LIN {X 0,Y 636.346,Z 292.016,A -85,B 0,C 180,E1 -5612.399,E2 -5612.399} C_VEL
LIN {X 0,Y 638.577,Z 243.118,A -85,B 0,C 180,E1 -5615.474,E2 -5615.474} C_VEL
LIN {X 0,Y 628.677,Z 217.087,A -85,B 0,C 180,E1 -5617.846,E2 -5617.846} C_VEL
LIN {X 0,Y 624.895,Z 207.391,A -85,B 0,C 180,E1 -5618.774,E2 -5618.774} C_VEL
LIN {X 0,Y 624.9,Z 207.391,A -85,B 0,C 180,E1 -5622.101,E2 -5622.101} C_VEL
LIN {X 0,Y 624.949,Z 207.381,A -85,B 0,C 180,E1 -5625.136,E2 -5625.136} C_VEL
LIN {X 0,Y 624.933,Z 207.387,A -85,B 0,C 180,E1 -5628.349,E2 -5628.349} C_VEL
LIN {X 0,Y 624.928,Z 207.584,A -85,B 0,C 180,E1 -5630.263,E2 -5630.263} C_VEL
LIN {X 0,Y 626.015,Z 210.6,A -85,B 0,C 180,E1 -5630.528,E2 -5630.528} C_VEL
LIN {X 0,Y 632.721,Z 226.25,A -85,B 0,C 180,E1 -5632.053,E2 -5632.053} C_VEL
LIN {X 0,Y 640.273,Z 245.58,A -85,B 0,C 180,E1 -5633.993,E2 -5633.993} C_VEL
LIN {X 0,Y 640.705,Z 247.691,A -85,B 0,C 180,E1 -5634.181,E2 -5634.181} C_VEL
LIN {X 0,Y 639.221,Z 289.191,A -85,B 0,C 180,E1 -5637.233,E2 -5637.233} C_VEL
LIN {X 0,Y 638.897,Z 318.308,A -85,B 0,C 180,E1 -5639.227,E2 -5639.227} C_VEL
LIN {X 0,Y 639.099,Z 324.989,A -85,B 0,C 180,E1 -5639.637,E2 -5639.637} C_VEL
LIN {X 0,Y 639.536,Z 329.306,A -85,B 0,C 180,E1 -5639.718,E2 -5639.718} C_VEL
LIN {X 0,Y 637.723,Z 440.539,A -85,B 0,C 180,E1 -5641.138,E2 -5641.138} C_VEL
LIN {X 0,Y 634.236,Z 617.38,A -85,B 0,C 180,E1 -5643.602,E2 -5643.602} C_VEL
LIN {X 0,Y 633.701,Z 640.001,A -85,B 0,C 180,E1 -5644.083,E2 -5644.083} C_VEL
LIN {X 0,Y 632.964,Z 662.226,A -85,B 0,C 180,E1 -5644.728,E2 -5644.728} C_VEL
LIN {X 0,Y 632.12,Z 684.246,A -85,B 0,C 180,E1 -5645.551,E2 -5645.551} C_VEL
LIN {X 0,Y 631.255,Z 703.32,A -85,B 0,C 180,E1 -5646.425,E2 -5646.425} C_VEL
LIN {X 0,Y 630.24,Z 722.986,A -85,B 0,C 180,E1 -5647.52,E2 -5647.52} C_VEL
LIN {X 0,Y 629.208,Z 740.926,A -85,B 0,C 180,E1 -5648.708,E2 -5648.708} C_VEL
LIN {X 0,Y 628.174,Z 758.568,A -85,B 0,C 180,E1 -5650.085,E2 -5650.085} C_VEL
LIN {X 0,Y 627.247,Z 774.118,A -85,B 0,C 180,E1 -5651.505,E2 -5651.505} C_VEL
LIN {X 0,Y 626.389,Z 788.139,A -85,B 0,C 180,E1 -5653.015,E2 -5653.015} C_VEL
LIN {X 0,Y 625.582,Z 802.216,A -85,B 0,C 180,E1 -5654.804,E2 -5654.804} C_VEL
LIN {X 0,Y 624.988,Z 813.341,A -85,B 0,C 180,E1 -5656.492,E2 -5656.492} C_VEL
LIN {X 0,Y 624.565,Z 822.244,A -85,B 0,C 180,E1 -5658.081,E2 -5658.081} C_VEL
LIN {X 0,Y 624.211,Z 832.3,A -85,B 0,C 180,E1 -5660.224,E2 -5660.224} C_VEL
LIN {X 0,Y 624.048,Z 838.961,A -85,B 0,C 180,E1 -5661.987,E2 -5661.987} C_VEL
LIN {X 0,Y 623.969,Z 843.988,A -85,B 0,C 180,E1 -5663.652,E2 -5663.652} C_VEL
LIN {X 0,Y 623.918,Z 847.629,A -85,B 0,C 180,E1 -5665.22,E2 -5665.22} C_VEL
LIN {X 0,Y 623.903,Z 850.253,A -85,B 0,C 180,E1 -5666.807,E2 -5666.807} C_VEL
LIN {X 0,Y 623.908,Z 851.807,A -85,B 0,C 180,E1 -5668.347,E2 -5668.347} C_VEL
LIN {X 0,Y 623.919,Z 852.393,A -85,B 0,C 180,E1 -5670,E2 -5670} C_VEL
LIN {X 0,Y 623.906,Z 851.865,A -85,B 0,C 180,E1 -5671.653,E2 -5671.653} C_VEL
LIN {X 0,Y 623.901,Z 850.34,A -85,B 0,C 180,E1 -5673.215,E2 -5673.215} C_VEL
LIN {X 0,Y 623.92,Z 847.804,A -85,B 0,C 180,E1 -5674.78,E2 -5674.78} C_VEL
LIN {X 0,Y 623.969,Z 844.223,A -85,B 0,C 180,E1 -5676.348,E2 -5676.348} C_VEL
LIN {X 0,Y 624.029,Z 839.56,A -85,B 0,C 180,E1 -5677.92,E2 -5677.92} C_VEL
LIN {X 0,Y 624.164,Z 833.767,A -85,B 0,C 180,E1 -5679.497,E2 -5679.497} C_VEL
LIN {X 0,Y 624.432,Z 825.538,A -85,B 0,C 180,E1 -5681.359,E2 -5681.359} C_VEL
LIN {X 0,Y 624.9,Z 815.025,A -85,B 0,C 180,E1 -5683.321,E2 -5683.321} C_VEL
LIN {X 0,Y 625.468,Z 804.166,A -85,B 0,C 180,E1 -5685.009,E2 -5685.009} C_VEL
LIN {X 0,Y 626.179,Z 791.739,A -85,B 0,C 180,E1 -5686.646,E2 -5686.646} C_VEL
LIN {X 0,Y 627.018,Z 777.74,A -85,B 0,C 180,E1 -5688.213,E2 -5688.213} C_VEL
LIN {X 0,Y 627.946,Z 762.367,A -85,B 0,C 180,E1 -5689.68,E2 -5689.68} C_VEL
LIN {X 0,Y 628.974,Z 745.456,A -85,B 0,C 180,E1 -5691.056,E2 -5691.056} C_VEL
LIN {X 0,Y 629.98,Z 727.417,A -85,B 0,C 180,E1 -5692.292,E2 -5692.292} C_VEL
LIN {X 0,Y 630.985,Z 708.54,A -85,B 0,C 180,E1 -5693.388,E2 -5693.388} C_VEL
LIN {X 0,Y 631.859,Z 689.995,A -85,B 0,C 180,E1 -5694.295,E2 -5694.295} C_VEL
LIN {X 0,Y 632.742,Z 669.051,A -85,B 0,C 180,E1 -5695.13,E2 -5695.13} C_VEL
LIN {X 0,Y 633.413,Z 648.623,A -85,B 0,C 180,E1 -5695.774,E2 -5695.774} C_VEL
LIN {X 0,Y 634.025,Z 626.542,A -85,B 0,C 180,E1 -5696.308,E2 -5696.308} C_VEL
LIN {X 0,Y 634.453,Z 605.1,A -85,B 0,C 180,E1 -5696.679,E2 -5696.679} C_VEL
LIN {X 0,Y 638.365,Z 407.202,A -85,B 0,C 180,E1 -5699.392,E2 -5699.392} C_VEL
LIN {X 0,Y 639.37,Z 326.363,A -85,B 0,C 180,E1 -5700.421,E2 -5700.421} C_VEL
LIN {X 0,Y 639.015,Z 324.152,A -85,B 0,C 180,E1 -5700.489,E2 -5700.489} C_VEL
LIN {X 0,Y 639.079,Z 296.354,A -85,B 0,C 180,E1 -5702.35,E2 -5702.35} C_VEL
LIN {X 0,Y 640.388,Z 256.622,A -85,B 0,C 180,E1 -5705.253,E2 -5705.253} C_VEL
LIN {X 0,Y 640.643,Z 246.721,A -85,B 0,C 180,E1 -5705.976,E2 -5705.976} C_VEL
LIN {X 0,Y 633.821,Z 228.869,A -85,B 0,C 180,E1 -5707.781,E2 -5707.781} C_VEL
LIN {X 0,Y 627.274,Z 213.434,A -85,B 0,C 180,E1 -5709.294,E2 -5709.294} C_VEL
LIN {X 0,Y 624.952,Z 207.388,A -85,B 0,C 180,E1 -5709.871,E2 -5709.871} C_VEL
LIN {X 0,Y 624.924,Z 207.385,A -85,B 0,C 180,E1 -5713.012,E2 -5713.012} C_VEL
LIN {X 0,Y 624.946,Z 207.377,A -85,B 0,C 180,E1 -5716.149,E2 -5716.149} C_VEL
LIN {X 0,Y 624.928,Z 207.382,A -85,B 0,C 180,E1 -5719.246,E2 -5719.246} C_VEL
LIN {X 0,Y 624.947,Z 207.376,A -85,B 0,C 180,E1 -5722.371,E2 -5722.371} C_VEL
LIN {X 0,Y 624.94,Z 207.389,A -85,B 0,C 180,E1 -5725.501,E2 -5725.501} C_VEL
LIN {X 0,Y 624.947,Z 207.379,A -85,B 0,C 180,E1 -5728.776,E2 -5728.776} C_VEL
LIN {X 0,Y 624.945,Z 207.373,A -85,B 0,C 180,E1 -5731.94,E2 -5731.94} C_VEL
LIN {X 0,Y 624.937,Z 207.381,A -85,B 0,C 180,E1 -5735.12,E2 -5735.12} C_VEL
LIN {X 0,Y 624.937,Z 207.383,A -85,B 0,C 180,E1 -5738.21,E2 -5738.21} C_VEL
LIN {X 0,Y 624.937,Z 207.371,A -85,B 0,C 180,E1 -5741.337,E2 -5741.337} C_VEL
LIN {X 0,Y 624.934,Z 207.381,A -85,B 0,C 180,E1 -5744.407,E2 -5744.407} C_VEL
LIN {X 0,Y 624.941,Z 207.366,A -85,B 0,C 180,E1 -5747.526,E2 -5747.526} C_VEL
LIN {X 0,Y 624.942,Z 207.38,A -85,B 0,C 180,E1 -5750.7,E2 -5750.7} C_VEL
LIN {X 0,Y 624.943,Z 207.365,A -85,B 0,C 180,E1 -5753.938,E2 -5753.938} C_VEL
LIN {X 0,Y 624.947,Z 207.38,A -85,B 0,C 180,E1 -5757.157,E2 -5757.157} C_VEL
LIN {X 0,Y 624.923,Z 207.363,A -85,B 0,C 180,E1 -5760.275,E2 -5760.275} C_VEL
LIN {X 0,Y 624.946,Z 207.381,A -85,B 0,C 180,E1 -5763.394,E2 -5763.394} C_VEL
LIN {X 0,Y 624.919,Z 207.364,A -85,B 0,C 180,E1 -5766.523,E2 -5766.523} C_VEL
LIN {X 0,Y 624.949,Z 207.381,A -85,B 0,C 180,E1 -5769.671,E2 -5769.671} C_VEL
LIN {X 0,Y 624.924,Z 207.382,A -85,B 0,C 180,E1 -5772.756,E2 -5772.756} C_VEL
LIN {X 0,Y 624.942,Z 207.385,A -85,B 0,C 180,E1 -5775.974,E2 -5775.974} C_VEL
LIN {X 0,Y 624.946,Z 207.377,A -85,B 0,C 180,E1 -5779.147,E2 -5779.147} C_VEL
LIN {X 0,Y 624.916,Z 207.388,A -85,B 0,C 180,E1 -5782.358,E2 -5782.358} C_VEL
LIN {X 0,Y 624.953,Z 207.381,A -85,B 0,C 180,E1 -5785.391,E2 -5785.391} C_VEL
LIN {X 0,Y 624.91,Z 207.385,A -85,B 0,C 180,E1 -5788.546,E2 -5788.546} C_VEL
LIN {X 0,Y 624.957,Z 207.381,A -85,B 0,C 180,E1 -5791.546,E2 -5791.546} C_VEL
LIN {X 0,Y 624.906,Z 207.388,A -85,B 0,C 180,E1 -5794.671,E2 -5794.671} C_VEL
LIN {X 0,Y 624.957,Z 207.38,A -85,B 0,C 180,E1 -5797.791,E2 -5797.791} C_VEL
LIN {X 0,Y 624.903,Z 207.389,A -85,B 0,C 180,E1 -5800.814,E2 -5800.814} C_VEL
LIN {X 0,Y 624.95,Z 207.462,A -85,B 0,C 180,E1 -5803.387,E2 -5803.387} C_VEL
LIN {X 0,Y 626.289,Z 210.904,A -85,B 0,C 180,E1 -5803.733,E2 -5803.733} C_VEL
LIN {X 0,Y 627.344,Z 212.887,A -85,B 0,C 180,E1 -5803.957,E2 -5803.957} C_VEL
LIN {X 0,Y 638.156,Z 234.423,A -85,B 0,C 180,E1 -5806.246,E2 -5806.246} C_VEL
LIN {X 0,Y 647.363,Z 253.935,A -85,B 0,C 180,E1 -5808.145,E2 -5808.145} C_VEL
LIN {X 0,Y 644.416,Z 304.648,A -85,B 0,C 180,E1 -5810.782,E2 -5810.782} C_VEL
LIN {X 0,Y 646.898,Z 323.157,A -85,B 0,C 180,E1 -5811.205,E2 -5811.205} C_VEL
LIN {X 0,Y 644.169,Z 514.087,A -85,B 0,C 180,E1 -5813.627,E2 -5813.627} C_VEL
LIN {X 0,Y 641.865,Z 692.934,A -85,B 0,C 180,E1 -5815.853,E2 -5815.853} C_VEL
LIN {X 0,Y 641.079,Z 718.1,A -85,B 0,C 180,E1 -5816.326,E2 -5816.326} C_VEL
LIN {X 0,Y 640.186,Z 739.868,A -85,B 0,C 180,E1 -5816.869,E2 -5816.869} C_VEL
LIN {X 0,Y 638.916,Z 765.321,A -85,B 0,C 180,E1 -5817.682,E2 -5817.682} C_VEL
LIN {X 0,Y 637.689,Z 787.238,A -85,B 0,C 180,E1 -5818.539,E2 -5818.539} C_VEL
LIN {X 0,Y 636.241,Z 810.546,A -85,B 0,C 180,E1 -5819.631,E2 -5819.631} C_VEL
LIN {X 0,Y 634.874,Z 830.591,A -85,B 0,C 180,E1 -5820.724,E2 -5820.724} C_VEL
LIN {X 0,Y 633.292,Z 852.909,A -85,B 0,C 180,E1 -5822.138,E2 -5822.138} C_VEL
LIN {X 0,Y 632.055,Z 867.818,A -85,B 0,C 180,E1 -5823.252,E2 -5823.252} C_VEL
LIN {X 0,Y 630.517,Z 886.159,A -85,B 0,C 180,E1 -5824.798,E2 -5824.798} C_VEL
LIN {X 0,Y 629.035,Z 903.822,A -85,B 0,C 180,E1 -5826.518,E2 -5826.518} C_VEL
LIN {X 0,Y 627.829,Z 919.315,A -85,B 0,C 180,E1 -5828.218,E2 -5828.218} C_VEL
LIN {X 0,Y 626.714,Z 934.515,A -85,B 0,C 180,E1 -5830.133,E2 -5830.133} C_VEL
LIN {X 0,Y 625.867,Z 947.149,A -85,B 0,C 180,E1 -5831.945,E2 -5831.945} C_VEL
LIN {X 0,Y 625.118,Z 960.283,A -85,B 0,C 180,E1 -5834.126,E2 -5834.126} C_VEL
LIN {X 0,Y 624.657,Z 970.018,A -85,B 0,C 180,E1 -5836.013,E2 -5836.013} C_VEL
LIN {X 0,Y 624.293,Z 979.836,A -85,B 0,C 180,E1 -5838.264,E2 -5838.264} C_VEL
LIN {X 0,Y 624.094,Z 986.816,A -85,B 0,C 180,E1 -5840.222,E2 -5840.222} C_VEL
LIN {X 0,Y 623.952,Z 993.243,A -85,B 0,C 180,E1 -5842.449,E2 -5842.449} C_VEL
LIN {X 0,Y 623.905,Z 997.655,A -85,B 0,C 180,E1 -5844.574,E2 -5844.574} C_VEL
LIN {X 0,Y 623.91,Z 1000.464,A -85,B 0,C 180,E1 -5846.509,E2 -5846.509} C_VEL
LIN {X 0,Y 623.909,Z 1002.214,A -85,B 0,C 180,E1 -5848.806,E2 -5848.806} C_VEL
LIN {X 0,Y 623.885,Z 1002.327,A -85,B 0,C 180,E1 -5850.735,E2 -5850.735} C_VEL
LIN {X 0,Y 623.889,Z 1001.292,A -85,B 0,C 180,E1 -5852.664,E2 -5852.664} C_VEL
LIN {X 0,Y 623.901,Z 998.451,A -85,B 0,C 180,E1 -5854.965,E2 -5854.965} C_VEL
LIN {X 0,Y 623.959,Z 994.689,A -85,B 0,C 180,E1 -5856.903,E2 -5856.903} C_VEL
LIN {X 0,Y 624.042,Z 988.934,A -85,B 0,C 180,E1 -5859.127,E2 -5859.127} C_VEL
LIN {X 0,Y 624.217,Z 981.602,A -85,B 0,C 180,E1 -5861.27,E2 -5861.27} C_VEL
LIN {X 0,Y 624.519,Z 973.532,A -85,B 0,C 180,E1 -5863.235,E2 -5863.235} C_VEL
LIN {X 0,Y 624.996,Z 962.86,A -85,B 0,C 180,E1 -5865.401,E2 -5865.401} C_VEL
LIN {X 0,Y 625.602,Z 951.969,A -85,B 0,C 180,E1 -5867.294,E2 -5867.294} C_VEL
LIN {X 0,Y 626.517,Z 937.317,A -85,B 0,C 180,E1 -5869.485,E2 -5869.485} C_VEL
LIN {X 0,Y 627.462,Z 924.012,A -85,B 0,C 180,E1 -5871.215,E2 -5871.215} C_VEL
LIN {X 0,Y 628.838,Z 906.301,A -85,B 0,C 180,E1 -5873.225,E2 -5873.225} C_VEL
LIN {X 0,Y 630.114,Z 890.795,A -85,B 0,C 180,E1 -5874.767,E2 -5874.767} C_VEL
LIN {X 0,Y 631.805,Z 870.854,A -85,B 0,C 180,E1 -5876.506,E2 -5876.506} C_VEL
LIN {X 0,Y 633.107,Z 855.309,A -85,B 0,C 180,E1 -5877.693,E2 -5877.693} C_VEL
LIN {X 0,Y 634.055,Z 841.543,A -85,B 0,C 180,E1 -5878.595,E2 -5878.595} C_VEL
LIN {X 0,Y 635.449,Z 820.222,A -85,B 0,C 180,E1 -5879.817,E2 -5879.817} C_VEL
LIN {X 0,Y 636.697,Z 797.901,A -85,B 0,C 180,E1 -5880.899,E2 -5880.899} C_VEL
LIN {X 0,Y 637.906,Z 775.285,A -85,B 0,C 180,E1 -5881.835,E2 -5881.835} C_VEL
LIN {X 0,Y 638.944,Z 751.93,A -85,B 0,C 180,E1 -5882.623,E2 -5882.623} C_VEL
LIN {X 0,Y 639.847,Z 727.921,A -85,B 0,C 180,E1 -5883.28,E2 -5883.28} C_VEL
LIN {X 0,Y 640.534,Z 703.096,A -85,B 0,C 180,E1 -5883.781,E2 -5883.781} C_VEL
LIN {X 0,Y 640.998,Z 677.434,A -85,B 0,C 180,E1 -5884.144,E2 -5884.144} C_VEL
LIN {X 0,Y 642.199,Z 471.258,A -85,B 0,C 180,E1 -5886.503,E2 -5886.503} C_VEL
LIN {X 0,Y 643.617,Z 320.826,A -85,B 0,C 180,E1 -5888.348,E2 -5888.348} C_VEL
LIN {X 0,Y 642.214,Z 312.028,A -85,B 0,C 180,E1 -5888.548,E2 -5888.548} C_VEL
LIN {X 0,Y 644.812,Z 281.295,A -85,B 0,C 180,E1 -5890.288,E2 -5890.288} C_VEL
LIN {X 0,Y 648.358,Z 254.707,A -85,B 0,C 180,E1 -5891.95,E2 -5891.95} C_VEL
LIN {X 0,Y 645.178,Z 246.171,A -85,B 0,C 180,E1 -5893.117,E2 -5893.117} C_VEL
LIN {X 0,Y 642.634,Z 240.116,A -85,B 0,C 180,E1 -5894.191,E2 -5894.191} C_VEL
LIN {X 0,Y 641.16,Z 236.75,A -85,B 0,C 180,E1 -5894.947,E2 -5894.947} C_VEL
LIN {X 0,Y 639.826,Z 233.597,A -85,B 0,C 180,E1 -5895.832,E2 -5895.832} C_VEL
LIN {X 0,Y 638.452,Z 230.647,A -85,B 0,C 180,E1 -5897.302,E2 -5897.302} C_VEL
LIN {X 0,Y 638.405,Z 229.859,A -85,B 0,C 180,E1 -5898.268,E2 -5898.268} C_VEL
LIN {X 0,Y 638.414,Z 231.106,A -85,B 0,C 180,E1 -5899.342,E2 -5899.342} C_VEL
LIN {X 0,Y 639.781,Z 233.899,A -85,B 0,C 180,E1 -5900.68,E2 -5900.68} C_VEL
LIN {X 0,Y 641.35,Z 238.172,A -85,B 0,C 180,E1 -5901.791,E2 -5901.791} C_VEL
LIN {X 0,Y 643.354,Z 243.746,A -85,B 0,C 180,E1 -5902.873,E2 -5902.873} C_VEL
LIN {X 0,Y 645.653,Z 251.249,A -85,B 0,C 180,E1 -5903.999,E2 -5903.999} C_VEL
LIN {X 0,Y 641.269,Z 281.594,A -85,B 0,C 180,E1 -5906.283,E2 -5906.283} C_VEL
LIN {X 0,Y 637.312,Z 322.129,A -85,B 0,C 180,E1 -5909.115,E2 -5909.115} C_VEL
LIN {X 0,Y 634.413,Z 366.282,A -85,B 0,C 180,E1 -5912.038,E2 -5912.038} C_VEL
LIN {X 0,Y 631.971,Z 416.413,A -85,B 0,C 180,E1 -5915.211,E2 -5915.211} C_VEL
LIN {X 0,Y 631.044,Z 441.253,A -85,B 0,C 180,E1 -5916.72,E2 -5916.72} C_VEL
LIN {X 0,Y 635.394,Z 479.453,A -85,B 0,C 180,E1 -5917.724,E2 -5917.724} C_VEL
LIN {X 0,Y 635.961,Z 488.203,A -85,B 0,C 180,E1 -5917.919,E2 -5917.919} C_VEL
LIN {X 0,Y 632.244,Z 601.48,A -85,B 0,C 180,E1 -5919.721,E2 -5919.721} C_VEL
LIN {X 0,Y 630.407,Z 684.522,A -85,B 0,C 180,E1 -5920.982,E2 -5920.982} C_VEL
LIN {X 0,Y 629.845,Z 705.803,A -85,B 0,C 180,E1 -5921.482,E2 -5921.482} C_VEL
LIN {X 0,Y 629.291,Z 724.826,A -85,B 0,C 180,E1 -5922.094,E2 -5922.094} C_VEL
LIN {X 0,Y 628.646,Z 743.951,A -85,B 0,C 180,E1 -5922.887,E2 -5922.887} C_VEL
LIN {X 0,Y 628.049,Z 760.98,A -85,B 0,C 180,E1 -5923.77,E2 -5923.77} C_VEL
LIN {X 0,Y 627.432,Z 777.32,A -85,B 0,C 180,E1 -5924.802,E2 -5924.802} C_VEL
LIN {X 0,Y 626.858,Z 791.603,A -85,B 0,C 180,E1 -5925.886,E2 -5925.886} C_VEL
LIN {X 0,Y 626.317,Z 804.831,A -85,B 0,C 180,E1 -5927.085,E2 -5927.085} C_VEL
LIN {X 0,Y 625.835,Z 816.839,A -85,B 0,C 180,E1 -5928.386,E2 -5928.386} C_VEL
LIN {X 0,Y 625.39,Z 828.124,A -85,B 0,C 180,E1 -5929.871,E2 -5929.871} C_VEL
LIN {X 0,Y 625.031,Z 837.79,A -85,B 0,C 180,E1 -5931.444,E2 -5931.444} C_VEL
LIN {X 0,Y 624.78,Z 845.408,A -85,B 0,C 180,E1 -5933.014,E2 -5933.014} C_VEL
LIN {X 0,Y 624.611,Z 851.521,A -85,B 0,C 180,E1 -5934.673,E2 -5934.673} C_VEL
LIN {X 0,Y 624.48,Z 855.819,A -85,B 0,C 180,E1 -5936.328,E2 -5936.328} C_VEL
LIN {X 0,Y 624.401,Z 858.528,A -85,B 0,C 180,E1 -5938.073,E2 -5938.073} C_VEL
LIN {X 0,Y 624.361,Z 859.436,A -85,B 0,C 180,E1 -5939.816,E2 -5939.816} C_VEL
LIN {X 0,Y 624.335,Z 858.578,A -85,B 0,C 180,E1 -5941.56,E2 -5941.56} C_VEL
LIN {X 0,Y 624.355,Z 855.951,A -85,B 0,C 180,E1 -5943.305,E2 -5943.305} C_VEL
LIN {X 0,Y 624.419,Z 851.496,A -85,B 0,C 180,E1 -5945.053,E2 -5945.053} C_VEL
LIN {X 0,Y 624.534,Z 845.462,A -85,B 0,C 180,E1 -5946.712,E2 -5946.712} C_VEL
LIN {X 0,Y 624.739,Z 837.497,A -85,B 0,C 180,E1 -5948.375,E2 -5948.375} C_VEL
LIN {X 0,Y 625.04,Z 827.956,A -85,B 0,C 180,E1 -5949.949,E2 -5949.949} C_VEL
LIN {X 0,Y 625.447,Z 816.489,A -85,B 0,C 180,E1 -5951.48,E2 -5951.48} C_VEL
LIN {X 0,Y 625.919,Z 804.267,A -85,B 0,C 180,E1 -5952.829,E2 -5952.829} C_VEL
LIN {X 0,Y 626.493,Z 790.059,A -85,B 0,C 180,E1 -5954.134,E2 -5954.134} C_VEL
LIN {X 0,Y 627.113,Z 775.015,A -85,B 0,C 180,E1 -5955.283,E2 -5955.283} C_VEL
LIN {X 0,Y 627.76,Z 758.503,A -85,B 0,C 180,E1 -5956.328,E2 -5956.328} C_VEL
LIN {X 0,Y 628.401,Z 741.33,A -85,B 0,C 180,E1 -5957.215,E2 -5957.215} C_VEL
LIN {X 0,Y 629.033,Z 723.273,A -85,B 0,C 180,E1 -5957.961,E2 -5957.961} C_VEL
LIN {X 0,Y 629.604,Z 703.456,A -85,B 0,C 180,E1 -5958.588,E2 -5958.588} C_VEL
LIN {X 0,Y 630.065,Z 683.762,A -85,B 0,C 180,E1 -5959.031,E2 -5959.031} C_VEL
LIN {X 0,Y 630.481,Z 653.884,A -85,B 0,C 180,E1 -5959.448,E2 -5959.448} C_VEL
LIN {X 0,Y 632.813,Z 483.695,A -85,B 0,C 180,E1 -5961.677,E2 -5961.677} C_VEL
LIN {X 0,Y 630.114,Z 460.538,A -85,B 0,C 180,E1 -5962.135,E2 -5962.135} C_VEL
LIN {X 0,Y 631.884,Z 406.271,A -85,B 0,C 180,E1 -5965.393,E2 -5965.393} C_VEL
LIN {X 0,Y 632.169,Z 397.972,A -85,B 0,C 180,E1 -5965.894,E2 -5965.894} C_VEL
LIN {X 0,Y 631.485,Z 391.743,A -85,B 0,C 180,E1 -5966.31,E2 -5966.31} C_VEL
LIN {X 0,Y 626.328,Z 376.015,A -85,B 0,C 180,E1 -5967.526,E2 -5967.526} C_VEL
LIN {X 0,Y 625.851,Z 370.657,A -85,B 0,C 180,E1 -5967.887,E2 -5967.887} C_VEL
LIN {X 0,Y 627.881,Z 321.996,A -85,B 0,C 180,E1 -5970.902,E2 -5970.902} C_VEL
LIN {X 0,Y 630.347,Z 269.288,A -85,B 0,C 180,E1 -5974.223,E2 -5974.223} C_VEL
LIN {X 0,Y 631.298,Z 245.645,A -85,B 0,C 180,E1 -5975.742,E2 -5975.742} C_VEL
LIN {X 0,Y 620.877,Z 218.382,A -85,B 0,C 180,E1 -5978.271,E2 -5978.271} C_VEL
LIN {X 0,Y 616.989,Z 208.38,A -85,B 0,C 180,E1 -5979.246,E2 -5979.246} C_VEL
LIN {X 0,Y 616.96,Z 208.381,A -85,B 0,C 180,E1 -5982.351,E2 -5982.351} C_VEL
LIN {X 0,Y 617.013,Z 208.37,A -85,B 0,C 180,E1 -5985.483,E2 -5985.483} C_VEL
LIN {X 0,Y 616.977,Z 208.375,A -85,B 0,C 180,E1 -5988.621,E2 -5988.621} C_VEL
LIN {X 0,Y 617.033,Z 208.453,A -85,B 0,C 180,E1 -5989.73,E2 -5989.73} C_VEL
LIN {X 0,Y 618.333,Z 211.922,A -85,B 0,C 180,E1 -5990.04,E2 -5990.04} C_VEL
LIN {X 0,Y 625.978,Z 229.789,A -85,B 0,C 180,E1 -5991.803,E2 -5991.803} C_VEL
LIN {X 0,Y 633.173,Z 248.32,A -85,B 0,C 180,E1 -5993.687,E2 -5993.687} C_VEL
LIN {X 0,Y 633.844,Z 251.207,A -85,B 0,C 180,E1 -5993.956,E2 -5993.956} C_VEL
LIN {X 0,Y 632.416,Z 295.085,A -85,B 0,C 180,E1 -5997.159,E2 -5997.159} C_VEL
LIN {X 0,Y 632.309,Z 325.01,A -85,B 0,C 180,E1 -5999.167,E2 -5999.167} C_VEL
LIN {X 0,Y 632.515,Z 327.844,A -85,B 0,C 180,E1 -5999.313,E2 -5999.313} C_VEL
LIN {X 0,Y 631.027,Z 428.42,A -85,B 0,C 180,E1 -6000.615,E2 -6000.615} C_VEL
LIN {X 0,Y 627.72,Z 572.114,A -85,B 0,C 180,E1 -6002.663,E2 -6002.663} C_VEL
LIN {X 0,Y 626.665,Z 621.823,A -85,B 0,C 180,E1 -6003.423,E2 -6003.423} C_VEL
LIN {X 0,Y 626.054,Z 644.64,A -85,B 0,C 180,E1 -6003.946,E2 -6003.946} C_VEL
LIN {X 0,Y 625.271,Z 666.522,A -85,B 0,C 180,E1 -6004.624,E2 -6004.624} C_VEL
LIN {X 0,Y 624.38,Z 687.651,A -85,B 0,C 180,E1 -6005.451,E2 -6005.451} C_VEL
LIN {X 0,Y 623.372,Z 708.562,A -85,B 0,C 180,E1 -6006.459,E2 -6006.459} C_VEL
LIN {X 0,Y 622.343,Z 727.705,A -85,B 0,C 180,E1 -6007.568,E2 -6007.568} C_VEL
LIN {X 0,Y 621.33,Z 745.237,A -85,B 0,C 180,E1 -6008.771,E2 -6008.771} C_VEL
LIN {X 0,Y 620.289,Z 761.787,A -85,B 0,C 180,E1 -6010.115,E2 -6010.115} C_VEL
LIN {X 0,Y 619.288,Z 777.907,A -85,B 0,C 180,E1 -6011.649,E2 -6011.649} C_VEL
LIN {X 0,Y 618.441,Z 791.683,A -85,B 0,C 180,E1 -6013.178,E2 -6013.178} C_VEL
LIN {X 0,Y 617.705,Z 804.058,A -85,B 0,C 180,E1 -6014.797,E2 -6014.797} C_VEL
LIN {X 0,Y 617.096,Z 815.114,A -85,B 0,C 180,E1 -6016.507,E2 -6016.507} C_VEL
LIN {X 0,Y 616.602,Z 825.387,A -85,B 0,C 180,E1 -6018.4,E2 -6018.4} C_VEL
LIN {X 0,Y 616.252,Z 834.032,A -85,B 0,C 180,E1 -6020.379,E2 -6020.379} C_VEL
LIN {X 0,Y 616.054,Z 840.215,A -85,B 0,C 180,E1 -6022.164,E2 -6022.164} C_VEL
LIN {X 0,Y 615.975,Z 844.61,A -85,B 0,C 180,E1 -6023.756,E2 -6023.756} C_VEL
LIN {X 0,Y 615.929,Z 848.876,A -85,B 0,C 180,E1 -6025.811,E2 -6025.811} C_VEL
LIN {X 0,Y 615.916,Z 851.625,A -85,B 0,C 180,E1 -6028.046,E2 -6028.046} C_VEL
LIN {X 0,Y 615.906,Z 852.387,A -85,B 0,C 180,E1 -6029.814,E2 -6029.814} C_VEL
LIN {X 0,Y 615.899,Z 851.978,A -85,B 0,C 180,E1 -6031.488,E2 -6031.488} C_VEL
LIN {X 0,Y 615.902,Z 850.572,A -85,B 0,C 180,E1 -6033.071,E2 -6033.071} C_VEL
LIN {X 0,Y 615.924,Z 848.154,A -85,B 0,C 180,E1 -6034.656,E2 -6034.656} C_VEL
LIN {X 0,Y 615.977,Z 844.374,A -85,B 0,C 180,E1 -6036.431,E2 -6036.431} C_VEL
LIN {X 0,Y 616.076,Z 839.628,A -85,B 0,C 180,E1 -6038.117,E2 -6038.117} C_VEL
LIN {X 0,Y 616.312,Z 832.537,A -85,B 0,C 180,E1 -6040.091,E2 -6040.091} C_VEL
LIN {X 0,Y 616.686,Z 823.437,A -85,B 0,C 180,E1 -6042.073,E2 -6042.073} C_VEL
LIN {X 0,Y 617.192,Z 813.408,A -85,B 0,C 180,E1 -6043.873,E2 -6043.873} C_VEL
LIN {X 0,Y 617.822,Z 801.948,A -85,B 0,C 180,E1 -6045.584,E2 -6045.584} C_VEL
LIN {X 0,Y 618.63,Z 788.345,A -85,B 0,C 180,E1 -6047.301,E2 -6047.301} C_VEL
LIN {X 0,Y 619.532,Z 774.136,A -85,B 0,C 180,E1 -6048.832,E2 -6048.832} C_VEL
LIN {X 0,Y 620.513,Z 758.369,A -85,B 0,C 180,E1 -6050.27,E2 -6050.27} C_VEL
LIN {X 0,Y 621.556,Z 741.112,A -85,B 0,C 180,E1 -6051.616,E2 -6051.616} C_VEL
LIN {X 0,Y 622.603,Z 723.132,A -85,B 0,C 180,E1 -6052.803,E2 -6052.803} C_VEL
LIN {X 0,Y 623.623,Z 703.837,A -85,B 0,C 180,E1 -6053.882,E2 -6053.882} C_VEL
LIN {X 0,Y 624.567,Z 683.722,A -85,B 0,C 180,E1 -6054.806,E2 -6054.806} C_VEL
LIN {X 0,Y 625.368,Z 663.257,A -85,B 0,C 180,E1 -6055.575,E2 -6055.575} C_VEL
LIN {X 0,Y 626.144,Z 641.208,A -85,B 0,C 180,E1 -6056.229,E2 -6056.229} C_VEL
LIN {X 0,Y 626.707,Z 619.44,A -85,B 0,C 180,E1 -6056.712,E2 -6056.712} C_VEL
LIN {X 0,Y 630.374,Z 458.135,A -85,B 0,C 180,E1 -6059.067,E2 -6059.067} C_VEL
LIN {X 0,Y 632.296,Z 356.258,A -85,B 0,C 180,E1 -6060.413,E2 -6060.413} C_VEL
LIN {X 0,Y 632.526,Z 327.84,A -85,B 0,C 180,E1 -6060.777,E2 -6060.777} C_VEL
LIN {X 0,Y 632.323,Z 325.004,A -85,B 0,C 180,E1 -6060.925,E2 -6060.925} C_VEL
LIN {X 0,Y 632.406,Z 297.282,A -85,B 0,C 180,E1 -6062.782,E2 -6062.782} C_VEL
LIN {X 0,Y 633.772,Z 254.797,A -85,B 0,C 180,E1 -6065.881,E2 -6065.881} C_VEL
LIN {X 0,Y 633.892,Z 250.34,A -85,B 0,C 180,E1 -6066.212,E2 -6066.212} C_VEL
LIN {X 0,Y 625.98,Z 229.699,A -85,B 0,C 180,E1 -6068.299,E2 -6068.299} C_VEL
LIN {X 0,Y 618.297,Z 211.831,A -85,B 0,C 180,E1 -6070.063,E2 -6070.063} C_VEL
LIN {X 0,Y 617.017,Z 208.37,A -85,B 0,C 180,E1 -6070.407,E2 -6070.407} C_VEL
LIN {X 0,Y 617.009,Z 208.367,A -85,B 0,C 180,E1 -6073.658,E2 -6073.658} C_VEL
LIN {X 0,Y 616.992,Z 208.368,A -85,B 0,C 180,E1 -6076.851,E2 -6076.851} C_VEL
LIN {X 0,Y 617.007,Z 208.367,A -85,B 0,C 180,E1 -6079.957,E2 -6079.957} C_VEL
LIN {X 0,Y 616.992,Z 208.364,A -85,B 0,C 180,E1 -6083.041,E2 -6083.041} C_VEL
LIN {X 0,Y 617.003,Z 208.365,A -85,B 0,C 180,E1 -6086.119,E2 -6086.119} C_VEL
LIN {X 0,Y 616.995,Z 208.374,A -85,B 0,C 180,E1 -6089.304,E2 -6089.304} C_VEL
LIN {X 0,Y 617.008,Z 208.365,A -85,B 0,C 180,E1 -6092.493,E2 -6092.493} C_VEL
LIN {X 0,Y 617.009,Z 208.359,A -85,B 0,C 180,E1 -6095.693,E2 -6095.693} C_VEL
LIN {X 0,Y 617.008,Z 208.367,A -85,B 0,C 180,E1 -6098.977,E2 -6098.977} C_VEL
LIN {X 0,Y 616.996,Z 208.355,A -85,B 0,C 180,E1 -6102.164,E2 -6102.164} C_VEL
LIN {X 0,Y 617.001,Z 208.372,A -85,B 0,C 180,E1 -6105.348,E2 -6105.348} C_VEL
LIN {X 0,Y 616.993,Z 208.359,A -85,B 0,C 180,E1 -6108.502,E2 -6108.502} C_VEL
LIN {X 0,Y 617.011,Z 208.373,A -85,B 0,C 180,E1 -6111.707,E2 -6111.707} C_VEL
LIN {X 0,Y 617.008,Z 208.354,A -85,B 0,C 180,E1 -6114.98,E2 -6114.98} C_VEL
LIN {X 0,Y 616.993,Z 208.37,A -85,B 0,C 180,E1 -6118.143,E2 -6118.143} C_VEL
LIN {X 0,Y 617.007,Z 208.349,A -85,B 0,C 180,E1 -6121.3,E2 -6121.3} C_VEL
LIN {X 0,Y 616.985,Z 208.371,A -85,B 0,C 180,E1 -6124.462,E2 -6124.462} C_VEL
LIN {X 0,Y 617.009,Z 208.349,A -85,B 0,C 180,E1 -6127.636,E2 -6127.636} C_VEL
LIN {X 0,Y 616.987,Z 208.371,A -85,B 0,C 180,E1 -6130.741,E2 -6130.741} C_VEL
LIN {X 0,Y 617.006,Z 208.376,A -85,B 0,C 180,E1 -6133.973,E2 -6133.973} C_VEL
LIN {X 0,Y 617.009,Z 208.37,A -85,B 0,C 180,E1 -6137.154,E2 -6137.154} C_VEL
LIN {X 0,Y 616.982,Z 208.375,A -85,B 0,C 180,E1 -6140.293,E2 -6140.293} C_VEL
LIN {X 0,Y 617.018,Z 208.372,A -85,B 0,C 180,E1 -6143.393,E2 -6143.393} C_VEL
LIN {X 0,Y 616.971,Z 208.37,A -85,B 0,C 180,E1 -6146.571,E2 -6146.571} C_VEL
LIN {X 0,Y 617.019,Z 208.369,A -85,B 0,C 180,E1 -6149.704,E2 -6149.704} C_VEL
LIN {X 0,Y 616.969,Z 208.376,A -85,B 0,C 180,E1 -6152.772,E2 -6152.772} C_VEL
LIN {X 0,Y 617.008,Z 208.37,A -85,B 0,C 180,E1 -6155.919,E2 -6155.919} C_VEL
LIN {X 0,Y 616.97,Z 208.376,A -85,B 0,C 180,E1 -6158.963,E2 -6158.963} C_VEL
LIN {X 0,Y 616.984,Z 208.374,A -85,B 0,C 180,E1 -6162.216,E2 -6162.216} C_VEL
LIN {X 0,Y 616.973,Z 208.473,A -85,B 0,C 180,E1 -6162.721,E2 -6162.721} C_VEL
LIN {X 0,Y 618.159,Z 211.679,A -85,B 0,C 180,E1 -6163.047,E2 -6163.047} C_VEL
LIN {X 0,Y 619.445,Z 213.94,A -85,B 0,C 180,E1 -6163.316,E2 -6163.316} C_VEL
LIN {X 0,Y 630.352,Z 235.7,A -85,B 0,C 180,E1 -6165.676,E2 -6165.676} C_VEL
LIN {X 0,Y 640.346,Z 256.314,A -85,B 0,C 180,E1 -6167.744,E2 -6167.744} C_VEL
LIN {X 0,Y 640.785,Z 257.643,A -85,B 0,C 180,E1 -6167.857,E2 -6167.857} C_VEL
LIN {X 0,Y 637.808,Z 305.28,A -85,B 0,C 180,E1 -6170.363,E2 -6170.363} C_VEL
LIN {X 0,Y 640.349,Z 324.485,A -85,B 0,C 180,E1 -6170.807,E2 -6170.807} C_VEL
LIN {X 0,Y 637.351,Z 514.536,A -85,B 0,C 180,E1 -6173.255,E2 -6173.255} C_VEL
LIN {X 0,Y 634.819,Z 693.056,A -85,B 0,C 180,E1 -6175.512,E2 -6175.512} C_VEL
LIN {X 0,Y 633.989,Z 718.022,A -85,B 0,C 180,E1 -6175.986,E2 -6175.986} C_VEL
LIN {X 0,Y 633.043,Z 739.755,A -85,B 0,C 180,E1 -6176.535,E2 -6176.535} C_VEL
LIN {X 0,Y 631.732,Z 764.586,A -85,B 0,C 180,E1 -6177.335,E2 -6177.335} C_VEL
LIN {X 0,Y 630.423,Z 786.292,A -85,B 0,C 180,E1 -6178.189,E2 -6178.189} C_VEL
LIN {X 0,Y 628.88,Z 810.034,A -85,B 0,C 180,E1 -6179.311,E2 -6179.311} C_VEL
LIN {X 0,Y 627.456,Z 829.744,A -85,B 0,C 180,E1 -6180.396,E2 -6180.396} C_VEL
LIN {X 0,Y 625.763,Z 852.12,A -85,B 0,C 180,E1 -6181.825,E2 -6181.825} C_VEL
LIN {X 0,Y 624.347,Z 870.25,A -85,B 0,C 180,E1 -6183.152,E2 -6183.152} C_VEL
LIN {X 0,Y 622.966,Z 887.246,A -85,B 0,C 180,E1 -6184.574,E2 -6184.574} C_VEL
LIN {X 0,Y 621.405,Z 904.515,A -85,B 0,C 180,E1 -6186.287,E2 -6186.287} C_VEL
LIN {X 0,Y 620.037,Z 920.984,A -85,B 0,C 180,E1 -6188.129,E2 -6188.129} C_VEL
LIN {X 0,Y 618.856,Z 935.914,A -85,B 0,C 180,E1 -6190.067,E2 -6190.067} C_VEL
LIN {X 0,Y 617.897,Z 949.659,A -85,B 0,C 180,E1 -6192.094,E2 -6192.094} C_VEL
LIN {X 0,Y 617.171,Z 961.311,A -85,B 0,C 180,E1 -6194.11,E2 -6194.11} C_VEL
LIN {X 0,Y 616.667,Z 971.394,A -85,B 0,C 180,E1 -6196.115,E2 -6196.115} C_VEL
LIN {X 0,Y 616.3,Z 980.543,A -85,B 0,C 180,E1 -6198.299,E2 -6198.299} C_VEL
LIN {X 0,Y 616.105,Z 987.119,A -85,B 0,C 180,E1 -6200.189,E2 -6200.189} C_VEL
LIN {X 0,Y 615.955,Z 993.45,A -85,B 0,C 180,E1 -6202.444,E2 -6202.444} C_VEL
LIN {X 0,Y 615.909,Z 997.654,A -85,B 0,C 180,E1 -6204.504,E2 -6204.504} C_VEL
LIN {X 0,Y 615.912,Z 1000.464,A -85,B 0,C 180,E1 -6206.463,E2 -6206.463} C_VEL
LIN {X 0,Y 615.909,Z 1002.214,A -85,B 0,C 180,E1 -6208.791,E2 -6208.791} C_VEL
LIN {X 0,Y 615.887,Z 1002.327,A -85,B 0,C 180,E1 -6210.744,E2 -6210.744} C_VEL
LIN {X 0,Y 615.888,Z 1001.291,A -85,B 0,C 180,E1 -6212.699,E2 -6212.699} C_VEL
LIN {X 0,Y 615.901,Z 998.451,A -85,B 0,C 180,E1 -6215.029,E2 -6215.029} C_VEL
LIN {X 0,Y 615.968,Z 994.689,A -85,B 0,C 180,E1 -6216.993,E2 -6216.993} C_VEL
LIN {X 0,Y 616.063,Z 988.934,A -85,B 0,C 180,E1 -6219.246,E2 -6219.246} C_VEL
LIN {X 0,Y 616.25,Z 981.601,A -85,B 0,C 180,E1 -6221.417,E2 -6221.417} C_VEL
LIN {X 0,Y 616.573,Z 973.534,A -85,B 0,C 180,E1 -6223.409,E2 -6223.409} C_VEL
LIN {X 0,Y 617.093,Z 962.859,A -85,B 0,C 180,E1 -6225.603,E2 -6225.603} C_VEL
LIN {X 0,Y 617.754,Z 951.968,A -85,B 0,C 180,E1 -6227.521,E2 -6227.521} C_VEL
LIN {X 0,Y 618.754,Z 937.315,A -85,B 0,C 180,E1 -6229.739,E2 -6229.739} C_VEL
LIN {X 0,Y 619.76,Z 924.072,A -85,B 0,C 180,E1 -6231.483,E2 -6231.483} C_VEL
LIN {X 0,Y 621.184,Z 907.148,A -85,B 0,C 180,E1 -6233.436,E2 -6233.436} C_VEL
LIN {X 0,Y 622.531,Z 891.808,A -85,B 0,C 180,E1 -6234.988,E2 -6234.988} C_VEL
LIN {X 0,Y 623.751,Z 877.634,A -85,B 0,C 180,E1 -6236.259,E2 -6236.259} C_VEL
LIN {X 0,Y 625.28,Z 857.186,A -85,B 0,C 180,E1 -6237.784,E2 -6237.784} C_VEL
LIN {X 0,Y 626.602,Z 838.163,A -85,B 0,C 180,E1 -6239.019,E2 -6239.019} C_VEL
LIN {X 0,Y 628.135,Z 814.525,A -85,B 0,C 180,E1 -6240.342,E2 -6240.342} C_VEL
LIN {X 0,Y 629.406,Z 793.652,A -85,B 0,C 180,E1 -6241.336,E2 -6241.336} C_VEL
LIN {X 0,Y 630.686,Z 768.887,A -85,B 0,C 180,E1 -6242.326,E2 -6242.326} C_VEL
LIN {X 0,Y 631.695,Z 746.627,A -85,B 0,C 180,E1 -6243.052,E2 -6243.052} C_VEL
LIN {X 0,Y 632.655,Z 721.058,A -85,B 0,C 180,E1 -6243.707,E2 -6243.707} C_VEL
LIN {X 0,Y 633.289,Z 698.869,A -85,B 0,C 180,E1 -6244.132,E2 -6244.132} C_VEL
LIN {X 0,Y 633.718,Z 665.184,A -85,B 0,C 180,E1 -6244.566,E2 -6244.566} C_VEL
LIN {X 0,Y 634.955,Z 479.261,A -85,B 0,C 180,E1 -6246.725,E2 -6246.725} C_VEL
LIN {X 0,Y 636.703,Z 327.978,A -85,B 0,C 180,E1 -6248.623,E2 -6248.623} C_VEL
LIN {X 0,Y 636.546,Z 320.962,A -85,B 0,C 180,E1 -6248.73,E2 -6248.73} C_VEL
LIN {X 0,Y 635.484,Z 314.12,A -85,B 0,C 180,E1 -6248.888,E2 -6248.888} C_VEL
LIN {X 0,Y 638.266,Z 285.583,A -85,B 0,C 180,E1 -6250.554,E2 -6250.554} C_VEL
LIN {X 0,Y 642.169,Z 259.764,A -85,B 0,C 180,E1 -6252.212,E2 -6252.212} C_VEL
LIN {X 0,Y 642.228,Z 258.59,A -85,B 0,C 180,E1 -6252.308,E2 -6252.308} C_VEL
LIN {X 0,Y 639.122,Z 249.943,A -85,B 0,C 180,E1 -6253.585,E2 -6253.585} C_VEL
LIN {X 0,Y 636.649,Z 243.671,A -85,B 0,C 180,E1 -6254.844,E2 -6254.844} C_VEL
LIN {X 0,Y 635.084,Z 239.999,A -85,B 0,C 180,E1 -6255.901,E2 -6255.901} C_VEL
LIN {X 0,Y 633.833,Z 237.204,A -85,B 0,C 180,E1 -6257.318,E2 -6257.318} C_VEL
LIN {X 0,Y 633.8,Z 236.401,A -85,B 0,C 180,E1 -6258.263,E2 -6258.263} C_VEL
LIN {X 0,Y 633.762,Z 237.707,A -85,B 0,C 180,E1 -6259.365,E2 -6259.365} C_VEL
LIN {X 0,Y 634.883,Z 240.241,A -85,B 0,C 180,E1 -6260.603,E2 -6260.603} C_VEL
LIN {X 0,Y 636.359,Z 244.575,A -85,B 0,C 180,E1 -6261.751,E2 -6261.751} C_VEL
LIN {X 0,Y 638.32,Z 250.537,A -85,B 0,C 180,E1 -6262.909,E2 -6262.909} C_VEL
LIN {X 0,Y 639.719,Z 255.46,A -85,B 0,C 180,E1 -6263.674,E2 -6263.674} C_VEL
LIN {X 0,Y 635.013,Z 284.273,A -85,B 0,C 180,E1 -6265.905,E2 -6265.905} C_VEL
LIN {X 0,Y 630.81,Z 322.111,A -85,B 0,C 180,E1 -6268.62,E2 -6268.62} C_VEL
LIN {X 0,Y 627.539,Z 365.868,A -85,B 0,C 180,E1 -6271.586,E2 -6271.586} C_VEL
LIN {X 0,Y 624.783,Z 415.762,A -85,B 0,C 180,E1 -6274.805,E2 -6274.805} C_VEL
LIN {X 0,Y 623.838,Z 438.254,A -85,B 0,C 180,E1 -6276.194,E2 -6276.194} C_VEL
LIN {X 0,Y 627.937,Z 474.401,A -85,B 0,C 180,E1 -6277.204,E2 -6277.204} C_VEL
LIN {X 0,Y 629.105,Z 489.006,A -85,B 0,C 180,E1 -6277.552,E2 -6277.552} C_VEL
LIN {X 0,Y 625.251,Z 593.403,A -85,B 0,C 180,E1 -6279.279,E2 -6279.279} C_VEL
LIN {X 0,Y 622.958,Z 685.281,A -85,B 0,C 180,E1 -6280.722,E2 -6280.722} C_VEL
LIN {X 0,Y 622.336,Z 706.835,A -85,B 0,C 180,E1 -6281.244,E2 -6281.244} C_VEL
LIN {X 0,Y 621.709,Z 726.543,A -85,B 0,C 180,E1 -6281.898,E2 -6281.898} C_VEL
LIN {X 0,Y 621.011,Z 745.815,A -85,B 0,C 180,E1 -6282.719,E2 -6282.719} C_VEL
LIN {X 0,Y 620.384,Z 762.755,A -85,B 0,C 180,E1 -6283.617,E2 -6283.617} C_VEL
LIN {X 0,Y 619.731,Z 778.89,A -85,B 0,C 180,E1 -6284.657,E2 -6284.657} C_VEL
LIN {X 0,Y 619.102,Z 793.493,A -85,B 0,C 180,E1 -6285.789,E2 -6285.789} C_VEL
LIN {X 0,Y 618.525,Z 806.716,A -85,B 0,C 180,E1 -6287.014,E2 -6287.014} C_VEL
LIN {X 0,Y 618.015,Z 818.608,A -85,B 0,C 180,E1 -6288.332,E2 -6288.332} C_VEL
LIN {X 0,Y 617.567,Z 829.154,A -85,B 0,C 180,E1 -6289.741,E2 -6289.741} C_VEL
LIN {X 0,Y 617.196,Z 838.337,A -85,B 0,C 180,E1 -6291.241,E2 -6291.241} C_VEL
LIN {X 0,Y 616.912,Z 846.081,A -85,B 0,C 180,E1 -6292.831,E2 -6292.831} C_VEL
LIN {X 0,Y 616.715,Z 852.453,A -85,B 0,C 180,E1 -6294.557,E2 -6294.557} C_VEL
LIN {X 0,Y 616.566,Z 856.904,A -85,B 0,C 180,E1 -6296.281,E2 -6296.281} C_VEL
LIN {X 0,Y 616.479,Z 859.501,A -85,B 0,C 180,E1 -6297.955,E2 -6297.955} C_VEL
LIN {X 0,Y 616.431,Z 860.478,A -85,B 0,C 180,E1 -6299.721,E2 -6299.721} C_VEL
LIN {X 0,Y 616.404,Z 859.673,A -85,B 0,C 180,E1 -6301.487,E2 -6301.487} C_VEL
LIN {X 0,Y 616.42,Z 857.088,A -85,B 0,C 180,E1 -6303.255,E2 -6303.255} C_VEL
LIN {X 0,Y 616.483,Z 852.666,A -85,B 0,C 180,E1 -6305.025,E2 -6305.025} C_VEL
LIN {X 0,Y 616.605,Z 846.665,A -85,B 0,C 180,E1 -6306.705,E2 -6306.705} C_VEL
LIN {X 0,Y 616.819,Z 838.736,A -85,B 0,C 180,E1 -6308.389,E2 -6308.389} C_VEL
LIN {X 0,Y 617.137,Z 829.244,A -85,B 0,C 180,E1 -6309.983,E2 -6309.983} C_VEL
LIN {X 0,Y 617.555,Z 818.24,A -85,B 0,C 180,E1 -6311.487,E2 -6311.487} C_VEL
LIN {X 0,Y 618.065,Z 805.716,A -85,B 0,C 180,E1 -6312.9,E2 -6312.9} C_VEL
LIN {X 0,Y 618.669,Z 791.613,A -85,B 0,C 180,E1 -6314.221,E2 -6314.221} C_VEL
LIN {X 0,Y 619.328,Z 776.469,A -85,B 0,C 180,E1 -6315.402,E2 -6315.402} C_VEL
LIN {X 0,Y 620.028,Z 759.586,A -85,B 0,C 180,E1 -6316.489,E2 -6316.489} C_VEL
LIN {X 0,Y 620.715,Z 742.199,A -85,B 0,C 180,E1 -6317.402,E2 -6317.402} C_VEL
LIN {X 0,Y 621.41,Z 723.397,A -85,B 0,C 180,E1 -6318.189,E2 -6318.189} C_VEL
LIN {X 0,Y 622.019,Z 703.449,A -85,B 0,C 180,E1 -6318.827,E2 -6318.827} C_VEL
LIN {X 0,Y 622.515,Z 683.599,A -85,B 0,C 180,E1 -6319.277,E2 -6319.277} C_VEL
LIN {X 0,Y 622.953,Z 653.668,A -85,B 0,C 180,E1 -6319.698,E2 -6319.698} C_VEL
LIN {X 0,Y 625.477,Z 484.522,A -85,B 0,C 180,E1 -6321.964,E2 -6321.964} C_VEL
LIN {X 0,Y 622.598,Z 459.59,A -85,B 0,C 180,E1 -6322.472,E2 -6322.472} C_VEL
LIN {X 0,Y 624.439,Z 406.912,A -85,B 0,C 180,E1 -6325.667,E2 -6325.667} C_VEL
LIN {X 0,Y 625.851,Z 370.657,A -85,B 0,C 180,E1 -6327.887,E2 -6327.887} C_VEL
LIN {X 0,Y 625.208,Z 364.456,A -85,B 0,C 180,E1 -6328.311,E2 -6328.311} C_VEL
LIN {X 0,Y 620.194,Z 348.83,A -85,B 0,C 180,E1 -6329.556,E2 -6329.556} C_VEL
LIN {X 0,Y 619.749,Z 343.494,A -85,B 0,C 180,E1 -6329.924,E2 -6329.924} C_VEL
LIN {X 0,Y 622.209,Z 291.194,A -85,B 0,C 180,E1 -6333.229,E2 -6333.229} C_VEL
LIN {X 0,Y 624.317,Z 248.989,A -85,B 0,C 180,E1 -6335.943,E2 -6335.943} C_VEL
LIN {X 0,Y 614.323,Z 222.767,A -85,B 0,C 180,E1 -6338.399,E2 -6338.399} C_VEL
LIN {X 0,Y 609.048,Z 209.364,A -85,B 0,C 180,E1 -6339.736,E2 -6339.736} C_VEL
LIN {X 0,Y 609.051,Z 209.365,A -85,B 0,C 180,E1 -6342.818,E2 -6342.818} C_VEL
LIN {X 0,Y 609.064,Z 209.364,A -85,B 0,C 180,E1 -6346.018,E2 -6346.018} C_VEL
LIN {X 0,Y 609.038,Z 209.363,A -85,B 0,C 180,E1 -6349.076,E2 -6349.076} C_VEL
LIN {X 0,Y 609.065,Z 209.524,A -85,B 0,C 180,E1 -6349.185,E2 -6349.185} C_VEL
LIN {X 0,Y 610.316,Z 212.754,A -85,B 0,C 180,E1 -6349.48,E2 -6349.48} C_VEL
LIN {X 0,Y 618.228,Z 230.9,A -85,B 0,C 180,E1 -6351.295,E2 -6351.295} C_VEL
LIN {X 0,Y 625.536,Z 249.642,A -85,B 0,C 180,E1 -6353.209,E2 -6353.209} C_VEL
LIN {X 0,Y 627.086,Z 254.149,A -85,B 0,C 180,E1 -6353.67,E2 -6353.67} C_VEL
LIN {X 0,Y 625.713,Z 298.975,A -85,B 0,C 180,E1 -6356.926,E2 -6356.926} C_VEL
LIN {X 0,Y 625.687,Z 327.356,A -85,B 0,C 180,E1 -6358.817,E2 -6358.817} C_VEL
LIN {X 0,Y 625.859,Z 330.298,A -85,B 0,C 180,E1 -6358.971,E2 -6358.971} C_VEL
LIN {X 0,Y 623.942,Z 436.328,A -85,B 0,C 180,E1 -6360.353,E2 -6360.353} C_VEL
LIN {X 0,Y 620.804,Z 560.124,A -85,B 0,C 180,E1 -6362.163,E2 -6362.163} C_VEL
LIN {X 0,Y 619.263,Z 622.776,A -85,B 0,C 180,E1 -6363.154,E2 -6363.154} C_VEL
LIN {X 0,Y 618.58,Z 645.235,A -85,B 0,C 180,E1 -6363.689,E2 -6363.689} C_VEL
LIN {X 0,Y 617.745,Z 666.569,A -85,B 0,C 180,E1 -6364.365,E2 -6364.365} C_VEL
LIN {X 0,Y 616.764,Z 688.482,A -85,B 0,C 180,E1 -6365.239,E2 -6365.239} C_VEL
LIN {X 0,Y 615.723,Z 709.232,A -85,B 0,C 180,E1 -6366.251,E2 -6366.251} C_VEL
LIN {X 0,Y 614.65,Z 728.503,A -85,B 0,C 180,E1 -6367.378,E2 -6367.378} C_VEL
LIN {X 0,Y 613.531,Z 747.331,A -85,B 0,C 180,E1 -6368.689,E2 -6368.689} C_VEL
LIN {X 0,Y 612.467,Z 763.817,A -85,B 0,C 180,E1 -6370.05,E2 -6370.05} C_VEL
LIN {X 0,Y 611.501,Z 778.996,A -85,B 0,C 180,E1 -6371.512,E2 -6371.512} C_VEL
LIN {X 0,Y 610.622,Z 792.738,A -85,B 0,C 180,E1 -6373.054,E2 -6373.054} C_VEL
LIN {X 0,Y 609.856,Z 805.133,A -85,B 0,C 180,E1 -6374.694,E2 -6374.694} C_VEL
LIN {X 0,Y 609.223,Z 816.24,A -85,B 0,C 180,E1 -6376.426,E2 -6376.426} C_VEL
LIN {X 0,Y 608.735,Z 826.087,A -85,B 0,C 180,E1 -6378.248,E2 -6378.248} C_VEL
LIN {X 0,Y 608.374,Z 834.479,A -85,B 0,C 180,E1 -6380.158,E2 -6380.158} C_VEL
LIN {X 0,Y 608.146,Z 841.105,A -85,B 0,C 180,E1 -6382.061,E2 -6382.061} C_VEL
LIN {X 0,Y 608.04,Z 846.258,A -85,B 0,C 180,E1 -6383.959,E2 -6383.959} C_VEL
LIN {X 0,Y 607.974,Z 850.366,A -85,B 0,C 180,E1 -6386.134,E2 -6386.134} C_VEL
LIN {X 0,Y 607.953,Z 852.525,A -85,B 0,C 180,E1 -6388.209,E2 -6388.209} C_VEL
LIN {X 0,Y 607.944,Z 853.145,A -85,B 0,C 180,E1 -6390.188,E2 -6390.188} C_VEL
LIN {X 0,Y 607.95,Z 852.331,A -85,B 0,C 180,E1 -6392.168,E2 -6392.168} C_VEL
LIN {X 0,Y 607.989,Z 849.591,A -85,B 0,C 180,E1 -6394.433,E2 -6394.433} C_VEL
LIN {X 0,Y 608.058,Z 845.335,A -85,B 0,C 180,E1 -6396.515,E2 -6396.515} C_VEL
LIN {X 0,Y 608.207,Z 839.338,A -85,B 0,C 180,E1 -6398.604,E2 -6398.604} C_VEL
LIN {X 0,Y 608.498,Z 831.712,A -85,B 0,C 180,E1 -6400.605,E2 -6400.605} C_VEL
LIN {X 0,Y 608.887,Z 822.613,A -85,B 0,C 180,E1 -6402.519,E2 -6402.519} C_VEL
LIN {X 0,Y 609.443,Z 812.13,A -85,B 0,C 180,E1 -6404.344,E2 -6404.344} C_VEL
LIN {X 0,Y 610.158,Z 800.248,A -85,B 0,C 180,E1 -6406.078,E2 -6406.078} C_VEL
LIN {X 0,Y 611.004,Z 786.675,A -85,B 0,C 180,E1 -6407.743,E2 -6407.743} C_VEL
LIN {X 0,Y 611.971,Z 771.582,A -85,B 0,C 180,E1 -6409.321,E2 -6409.321} C_VEL
LIN {X 0,Y 612.988,Z 755.781,A -85,B 0,C 180,E1 -6410.73,E2 -6410.73} C_VEL
LIN {X 0,Y 614.111,Z 737.807,A -85,B 0,C 180,E1 -6412.093,E2 -6412.093} C_VEL
LIN {X 0,Y 615.156,Z 719.448,A -85,B 0,C 180,E1 -6413.265,E2 -6413.265} C_VEL
LIN {X 0,Y 616.177,Z 700.451,A -85,B 0,C 180,E1 -6414.29,E2 -6414.29} C_VEL
LIN {X 0,Y 617.171,Z 679.815,A -85,B 0,C 180,E1 -6415.22,E2 -6415.22} C_VEL
LIN {X 0,Y 618.091,Z 658.548,A -85,B 0,C 180,E1 -6416.002,E2 -6416.002} C_VEL
LIN {X 0,Y 618.873,Z 636.219,A -85,B 0,C 180,E1 -6416.638,E2 -6416.638} C_VEL
LIN {X 0,Y 619.458,Z 614.138,A -85,B 0,C 180,E1 -6417.09,E2 -6417.09} C_VEL
LIN {X 0,Y 623.142,Z 469.818,A -85,B 0,C 180,E1 -6419.266,E2 -6419.266} C_VEL
LIN {X 0,Y 625.193,Z 372.412,A -85,B 0,C 180,E1 -6420.588,E2 -6420.588} C_VEL
LIN {X 0,Y 625.761,Z 329.323,A -85,B 0,C 180,E1 -6421.152,E2 -6421.152} C_VEL
LIN {X 0,Y 625.683,Z 301.876,A -85,B 0,C 180,E1 -6422.966,E2 -6422.966} C_VEL
LIN {X 0,Y 626.834,Z 263.084,A -85,B 0,C 180,E1 -6425.776,E2 -6425.776} C_VEL
LIN {X 0,Y 627.148,Z 254.032,A -85,B 0,C 180,E1 -6426.439,E2 -6426.439} C_VEL
LIN {X 0,Y 619.261,Z 233.33,A -85,B 0,C 180,E1 -6428.554,E2 -6428.554} C_VEL
LIN {X 0,Y 611.939,Z 216.296,A -85,B 0,C 180,E1 -6430.265,E2 -6430.265} C_VEL
LIN {X 0,Y 609.278,Z 210.504,A -85,B 0,C 180,E1 -6430.839,E2 -6430.839} C_VEL
LIN {X 0,Y 609.046,Z 209.357,A -85,B 0,C 180,E1 -6430.957,E2 -6430.957} C_VEL
LIN {X 0,Y 609.071,Z 209.359,A -85,B 0,C 180,E1 -6434.112,E2 -6434.112} C_VEL
LIN {X 0,Y 609.052,Z 209.361,A -85,B 0,C 180,E1 -6437.31,E2 -6437.31} C_VEL
LIN {X 0,Y 609.076,Z 209.359,A -85,B 0,C 180,E1 -6440.556,E2 -6440.556} C_VEL
LIN {X 0,Y 609.07,Z 209.355,A -85,B 0,C 180,E1 -6443.872,E2 -6443.872} C_VEL
LIN {X 0,Y 609.053,Z 209.349,A -85,B 0,C 180,E1 -6447.084,E2 -6447.084} C_VEL
LIN {X 0,Y 609.064,Z 209.355,A -85,B 0,C 180,E1 -6450.17,E2 -6450.17} C_VEL
LIN {X 0,Y 609.061,Z 209.358,A -85,B 0,C 180,E1 -6453.373,E2 -6453.373} C_VEL
LIN {X 0,Y 609.069,Z 209.339,A -85,B 0,C 180,E1 -6456.591,E2 -6456.591} C_VEL
LIN {X 0,Y 609.069,Z 209.357,A -85,B 0,C 180,E1 -6459.89,E2 -6459.89} C_VEL
LIN {X 0,Y 609.061,Z 209.347,A -85,B 0,C 180,E1 -6463.158,E2 -6463.158} C_VEL
LIN {X 0,Y 609.056,Z 209.35,A -85,B 0,C 180,E1 -6466.229,E2 -6466.229} C_VEL
LIN {X 0,Y 609.064,Z 209.35,A -85,B 0,C 180,E1 -6469.405,E2 -6469.405} C_VEL
LIN {X 0,Y 609.055,Z 209.35,A -85,B 0,C 180,E1 -6472.565,E2 -6472.565} C_VEL
LIN {X 0,Y 609.068,Z 209.354,A -85,B 0,C 180,E1 -6475.858,E2 -6475.858} C_VEL
LIN {X 0,Y 609.075,Z 209.352,A -85,B 0,C 180,E1 -6479.059,E2 -6479.059} C_VEL
LIN {X 0,Y 609.049,Z 209.36,A -85,B 0,C 180,E1 -6482.258,E2 -6482.258} C_VEL
LIN {X 0,Y 609.07,Z 209.357,A -85,B 0,C 180,E1 -6485.464,E2 -6485.464} C_VEL
LIN {X 0,Y 609.043,Z 209.355,A -85,B 0,C 180,E1 -6488.592,E2 -6488.592} C_VEL
LIN {X 0,Y 609.073,Z 209.365,A -85,B 0,C 180,E1 -6491.842,E2 -6491.842} C_VEL
LIN {X 0,Y 609.06,Z 209.357,A -85,B 0,C 180,E1 -6495.034,E2 -6495.034} C_VEL
LIN {X 0,Y 609.045,Z 209.36,A -85,B 0,C 180,E1 -6498.275,E2 -6498.275} C_VEL
LIN {X 0,Y 609.077,Z 209.358,A -85,B 0,C 180,E1 -6501.438,E2 -6501.438} C_VEL
LIN {X 0,Y 609.035,Z 209.363,A -85,B 0,C 180,E1 -6504.559,E2 -6504.559} C_VEL
LIN {X 0,Y 609.076,Z 209.359,A -85,B 0,C 180,E1 -6507.684,E2 -6507.684} C_VEL
LIN {X 0,Y 609.031,Z 209.365,A -85,B 0,C 180,E1 -6510.703,E2 -6510.703} C_VEL
LIN {X 0,Y 609.076,Z 209.358,A -85,B 0,C 180,E1 -6513.832,E2 -6513.832} C_VEL
LIN {X 0,Y 609.033,Z 209.365,A -85,B 0,C 180,E1 -6516.934,E2 -6516.934} C_VEL
LIN {X 0,Y 609.048,Z 209.36,A -85,B 0,C 180,E1 -6520.181,E2 -6520.181} C_VEL
LIN {X 0,Y 609.081,Z 209.513,A -85,B 0,C 180,E1 -6522.051,E2 -6522.051} C_VEL
LIN {X 0,Y 610.077,Z 212.43,A -85,B 0,C 180,E1 -6522.347,E2 -6522.347} C_VEL
LIN {X 0,Y 611.359,Z 214.646,A -85,B 0,C 180,E1 -6522.618,E2 -6522.618} C_VEL
LIN {X 0,Y 622.163,Z 236.027,A -85,B 0,C 180,E1 -6525.002,E2 -6525.002} C_VEL
LIN {X 0,Y 632.92,Z 258.196,A -85,B 0,C 180,E1 -6527.275,E2 -6527.275} C_VEL
LIN {X 0,Y 634.211,Z 261.306,A -85,B 0,C 180,E1 -6527.563,E2 -6527.563} C_VEL
LIN {X 0,Y 631.23,Z 306.025,A -85,B 0,C 180,E1 -6529.939,E2 -6529.939} C_VEL
LIN {X 0,Y 633.831,Z 325.862,A -85,B 0,C 180,E1 -6530.402,E2 -6530.402} C_VEL
LIN {X 0,Y 629.969,Z 550.131,A -85,B 0,C 180,E1 -6533.333,E2 -6533.333} C_VEL
LIN {X 0,Y 627.801,Z 692.847,A -85,B 0,C 180,E1 -6535.157,E2 -6535.157} C_VEL
LIN {X 0,Y 626.927,Z 717.852,A -85,B 0,C 180,E1 -6535.637,E2 -6535.637} C_VEL
LIN {X 0,Y 625.933,Z 739.401,A -85,B 0,C 180,E1 -6536.188,E2 -6536.188} C_VEL
LIN {X 0,Y 624.507,Z 764.89,A -85,B 0,C 180,E1 -6537.018,E2 -6537.018} C_VEL
LIN {X 0,Y 623.063,Z 787.478,A -85,B 0,C 180,E1 -6537.923,E2 -6537.923} C_VEL
LIN {X 0,Y 621.444,Z 810.737,A -85,B 0,C 180,E1 -6539.047,E2 -6539.047} C_VEL
LIN {X 0,Y 619.86,Z 831.434,A -85,B 0,C 180,E1 -6540.209,E2 -6540.209} C_VEL
LIN {X 0,Y 618.139,Z 852.729,A -85,B 0,C 180,E1 -6541.604,E2 -6541.604} C_VEL
LIN {X 0,Y 616.56,Z 872.034,A -85,B 0,C 180,E1 -6543.046,E2 -6543.046} C_VEL
LIN {X 0,Y 614.929,Z 891.256,A -85,B 0,C 180,E1 -6544.699,E2 -6544.699} C_VEL
LIN {X 0,Y 613.765,Z 905.347,A -85,B 0,C 180,E1 -6546.068,E2 -6546.068} C_VEL
LIN {X 0,Y 612.386,Z 920.985,A -85,B 0,C 180,E1 -6547.841,E2 -6547.841} C_VEL
LIN {X 0,Y 611.099,Z 935.912,A -85,B 0,C 180,E1 -6549.803,E2 -6549.803} C_VEL
LIN {X 0,Y 610.065,Z 949.661,A -85,B 0,C 180,E1 -6551.856,E2 -6551.856} C_VEL
LIN {X 0,Y 609.286,Z 961.309,A -85,B 0,C 180,E1 -6553.898,E2 -6553.898} C_VEL
LIN {X 0,Y 608.741,Z 971.393,A -85,B 0,C 180,E1 -6555.931,E2 -6555.931} C_VEL
LIN {X 0,Y 608.345,Z 980.543,A -85,B 0,C 180,E1 -6558.144,E2 -6558.144} C_VEL
LIN {X 0,Y 608.116,Z 987.422,A -85,B 0,C 180,E1 -6560.154,E2 -6560.154} C_VEL
LIN {X 0,Y 607.957,Z 993.863,A -85,B 0,C 180,E1 -6562.535,E2 -6562.535} C_VEL
LIN {X 0,Y 607.909,Z 997.814,A -85,B 0,C 180,E1 -6564.526,E2 -6564.526} C_VEL
LIN {X 0,Y 607.905,Z 1000.689,A -85,B 0,C 180,E1 -6566.605,E2 -6566.605} C_VEL
LIN {X 0,Y 607.902,Z 1002.259,A -85,B 0,C 180,E1 -6568.963,E2 -6568.963} C_VEL
LIN {X 0,Y 607.89,Z 1002.304,A -85,B 0,C 180,E1 -6570.848,E2 -6570.848} C_VEL
LIN {X 0,Y 607.887,Z 1001.087,A -85,B 0,C 180,E1 -6573.017,E2 -6573.017} C_VEL
LIN {X 0,Y 607.903,Z 998.132,A -85,B 0,C 180,E1 -6575.285,E2 -6575.285} C_VEL
LIN {X 0,Y 607.963,Z 994.482,A -85,B 0,C 180,E1 -6577.18,E2 -6577.18} C_VEL
LIN {X 0,Y 608.096,Z 988.633,A -85,B 0,C 180,E1 -6579.464,E2 -6579.464} C_VEL
LIN {X 0,Y 608.289,Z 981.6,A -85,B 0,C 180,E1 -6581.569,E2 -6581.569} C_VEL
LIN {X 0,Y 608.632,Z 973.534,A -85,B 0,C 180,E1 -6583.587,E2 -6583.587} C_VEL
LIN {X 0,Y 609.198,Z 962.857,A -85,B 0,C 180,E1 -6585.811,E2 -6585.811} C_VEL
LIN {X 0,Y 609.898,Z 952.127,A -85,B 0,C 180,E1 -6587.727,E2 -6587.727} C_VEL
LIN {X 0,Y 610.945,Z 938.013,A -85,B 0,C 180,E1 -6589.902,E2 -6589.902} C_VEL
LIN {X 0,Y 612.012,Z 924.841,A -85,B 0,C 180,E1 -6591.668,E2 -6591.668} C_VEL
LIN {X 0,Y 613.526,Z 908.15,A -85,B 0,C 180,E1 -6593.636,E2 -6593.636} C_VEL
LIN {X 0,Y 614.591,Z 895.26,A -85,B 0,C 180,E1 -6594.921,E2 -6594.921} C_VEL
LIN {X 0,Y 615.854,Z 878.985,A -85,B 0,C 180,E1 -6596.334,E2 -6596.334} C_VEL
LIN {X 0,Y 617.384,Z 859.422,A -85,B 0,C 180,E1 -6597.836,E2 -6597.836} C_VEL
LIN {X 0,Y 618.881,Z 838.77,A -85,B 0,C 180,E1 -6599.204,E2 -6599.204} C_VEL
LIN {X 0,Y 620.437,Z 816.025,A -85,B 0,C 180,E1 -6600.508,E2 -6600.508} C_VEL
LIN {X 0,Y 621.785,Z 794.8,A -85,B 0,C 180,E1 -6601.538,E2 -6601.538} C_VEL
LIN {X 0,Y 623.109,Z 770.964,A -85,B 0,C 180,E1 -6602.518,E2 -6602.518} C_VEL
LIN {X 0,Y 624.156,Z 748.988,A -85,B 0,C 180,E1 -6603.255,E2 -6603.255} C_VEL
LIN {X 0,Y 625.146,Z 724.43,A -85,B 0,C 180,E1 -6603.917,E2 -6603.917} C_VEL
LIN {X 0,Y 625.846,Z 701.437,A -85,B 0,C 180,E1 -6604.375,E2 -6604.375} C_VEL
LIN {X 0,Y 626.312,Z 674.817,A -85,B 0,C 180,E1 -6604.748,E2 -6604.748} C_VEL
LIN {X 0,Y 627.717,Z 491.439,A -85,B 0,C 180,E1 -6606.906,E2 -6606.906} C_VEL
LIN {X 0,Y 629.694,Z 341.468,A -85,B 0,C 180,E1 -6608.827,E2 -6608.827} C_VEL
LIN {X 0,Y 629.797,Z 322.462,A -85,B 0,C 180,E1 -6609.099,E2 -6609.099} C_VEL
LIN {X 0,Y 628.881,Z 316.063,A -85,B 0,C 180,E1 -6609.257,E2 -6609.257} C_VEL
LIN {X 0,Y 632.1,Z 287.734,A -85,B 0,C 180,E1 -6610.971,E2 -6610.971} C_VEL
LIN {X 0,Y 636.352,Z 263.054,A -85,B 0,C 180,E1 -6612.612,E2 -6612.612} C_VEL
LIN {X 0,Y 633.88,Z 255.73,A -85,B 0,C 180,E1 -6613.742,E2 -6613.742} C_VEL
LIN {X 0,Y 631.684,Z 249.812,A -85,B 0,C 180,E1 -6614.963,E2 -6614.963} C_VEL
LIN {X 0,Y 630.151,Z 246.148,A -85,B 0,C 180,E1 -6616.086,E2 -6616.086} C_VEL
LIN {X 0,Y 629.209,Z 243.68,A -85,B 0,C 180,E1 -6617.393,E2 -6617.393} C_VEL
LIN {X 0,Y 629.197,Z 242.962,A -85,B 0,C 180,E1 -6618.323,E2 -6618.323} C_VEL
LIN {X 0,Y 629.247,Z 244.845,A -85,B 0,C 180,E1 -6619.706,E2 -6619.706} C_VEL
LIN {X 0,Y 630.015,Z 246.442,A -85,B 0,C 180,E1 -6620.474,E2 -6620.474} C_VEL
LIN {X 0,Y 631.27,Z 250.62,A -85,B 0,C 180,E1 -6621.633,E2 -6621.633} C_VEL
LIN {X 0,Y 633.282,Z 257.321,A -85,B 0,C 180,E1 -6622.945,E2 -6622.945} C_VEL
LIN {X 0,Y 633.886,Z 259.837,A -85,B 0,C 180,E1 -6623.341,E2 -6623.341} C_VEL
LIN {X 0,Y 628.956,Z 286.56,A -85,B 0,C 180,E1 -6625.476,E2 -6625.476} C_VEL
LIN {X 0,Y 624.452,Z 322.133,A -85,B 0,C 180,E1 -6628.102,E2 -6628.102} C_VEL
LIN {X 0,Y 620.823,Z 364.601,A -85,B 0,C 180,E1 -6631.054,E2 -6631.054} C_VEL
LIN {X 0,Y 617.801,Z 412.201,A -85,B 0,C 180,E1 -6634.191,E2 -6634.191} C_VEL
LIN {X 0,Y 616.724,Z 435.374,A -85,B 0,C 180,E1 -6635.653,E2 -6635.653} C_VEL
LIN {X 0,Y 620.799,Z 471.664,A -85,B 0,C 180,E1 -6636.717,E2 -6636.717} C_VEL
LIN {X 0,Y 622.255,Z 490.045,A -85,B 0,C 180,E1 -6637.182,E2 -6637.182} C_VEL
LIN {X 0,Y 617.805,Z 602.169,A -85,B 0,C 180,E1 -6639.092,E2 -6639.092} C_VEL
LIN {X 0,Y 615.556,Z 685.269,A -85,B 0,C 180,E1 -6640.439,E2 -6640.439} C_VEL
LIN {X 0,Y 614.874,Z 706.996,A -85,B 0,C 180,E1 -6640.974,E2 -6640.974} C_VEL
LIN {X 0,Y 614.2,Z 726.92,A -85,B 0,C 180,E1 -6641.641,E2 -6641.641} C_VEL
LIN {X 0,Y 613.468,Z 745.927,A -85,B 0,C 180,E1 -6642.457,E2 -6642.457} C_VEL
LIN {X 0,Y 612.789,Z 762.834,A -85,B 0,C 180,E1 -6643.36,E2 -6643.36} C_VEL
LIN {X 0,Y 612.093,Z 779.124,A -85,B 0,C 180,E1 -6644.412,E2 -6644.412} C_VEL
LIN {X 0,Y 611.422,Z 793.892,A -85,B 0,C 180,E1 -6645.558,E2 -6645.558} C_VEL
LIN {X 0,Y 610.824,Z 806.763,A -85,B 0,C 180,E1 -6646.752,E2 -6646.752} C_VEL
LIN {X 0,Y 610.268,Z 818.84,A -85,B 0,C 180,E1 -6648.086,E2 -6648.086} C_VEL
LIN {X 0,Y 609.752,Z 830.204,A -85,B 0,C 180,E1 -6649.608,E2 -6649.608} C_VEL
LIN {X 0,Y 609.35,Z 839.415,A -85,B 0,C 180,E1 -6651.127,E2 -6651.127} C_VEL
LIN {X 0,Y 609.04,Z 847.181,A -85,B 0,C 180,E1 -6652.738,E2 -6652.738} C_VEL
LIN {X 0,Y 608.824,Z 853.415,A -85,B 0,C 180,E1 -6654.439,E2 -6654.439} C_VEL
LIN {X 0,Y 608.661,Z 857.803,A -85,B 0,C 180,E1 -6656.138,E2 -6656.138} C_VEL
LIN {X 0,Y 608.554,Z 860.573,A -85,B 0,C 180,E1 -6657.928,E2 -6657.928} C_VEL
LIN {X 0,Y 608.499,Z 861.523,A -85,B 0,C 180,E1 -6659.718,E2 -6659.718} C_VEL
LIN {X 0,Y 608.468,Z 860.678,A -85,B 0,C 180,E1 -6661.507,E2 -6661.507} C_VEL
LIN {X 0,Y 608.485,Z 858.041,A -85,B 0,C 180,E1 -6663.297,E2 -6663.297} C_VEL
LIN {X 0,Y 608.548,Z 853.835,A -85,B 0,C 180,E1 -6664.996,E2 -6664.996} C_VEL
LIN {X 0,Y 608.676,Z 847.868,A -85,B 0,C 180,E1 -6666.698,E2 -6666.698} C_VEL
LIN {X 0,Y 608.9,Z 839.974,A -85,B 0,C 180,E1 -6668.404,E2 -6668.404} C_VEL
LIN {X 0,Y 609.235,Z 830.491,A -85,B 0,C 180,E1 -6670.024,E2 -6670.024} C_VEL
LIN {X 0,Y 609.671,Z 819.569,A -85,B 0,C 180,E1 -6671.542,E2 -6671.542} C_VEL
LIN {X 0,Y 610.207,Z 807.122,A -85,B 0,C 180,E1 -6672.973,E2 -6672.973} C_VEL
LIN {X 0,Y 610.844,Z 793.148,A -85,B 0,C 180,E1 -6674.31,E2 -6674.31} C_VEL
LIN {X 0,Y 611.562,Z 777.487,A -85,B 0,C 180,E1 -6675.553,E2 -6675.553} C_VEL
LIN {X 0,Y 612.301,Z 760.669,A -85,B 0,C 180,E1 -6676.654,E2 -6676.654} C_VEL
LIN {X 0,Y 613.009,Z 743.732,A -85,B 0,C 180,E1 -6677.563,E2 -6677.563} C_VEL
LIN {X 0,Y 613.709,Z 726.099,A -85,B 0,C 180,E1 -6678.328,E2 -6678.328} C_VEL
LIN {X 0,Y 614.339,Z 706.874,A -85,B 0,C 180,E1 -6678.975,E2 -6678.975} C_VEL
LIN {X 0,Y 614.884,Z 687.11,A -85,B 0,C 180,E1 -6679.457,E2 -6679.457} C_VEL
LIN {X 0,Y 615.326,Z 663.198,A -85,B 0,C 180,E1 -6679.831,E2 -6679.831} C_VEL
LIN {X 0,Y 618.192,Z 485.565,A -85,B 0,C 180,E1 -6682.256,E2 -6682.256} C_VEL
LIN {X 0,Y 615.087,Z 459.086,A -85,B 0,C 180,E1 -6682.789,E2 -6682.789} C_VEL
LIN {X 0,Y 617.03,Z 406.969,A -85,B 0,C 180,E1 -6685.983,E2 -6685.983} C_VEL
LIN {X 0,Y 619.24,Z 355.289,A -85,B 0,C 180,E1 -6689.186,E2 -6689.186} C_VEL
LIN {X 0,Y 619.749,Z 343.494,A -85,B 0,C 180,E1 -6689.924,E2 -6689.924} C_VEL
LIN {X 0,Y 619.14,Z 337.327,A -85,B 0,C 180,E1 -6690.356,E2 -6690.356} C_VEL
LIN {X 0,Y 614.246,Z 321.833,A -85,B 0,C 180,E1 -6691.63,E2 -6691.63} C_VEL
LIN {X 0,Y 613.838,Z 316.525,A -85,B 0,C 180,E1 -6692.005,E2 -6692.005} C_VEL
LIN {X 0,Y 616.449,Z 266.722,A -85,B 0,C 180,E1 -6695.214,E2 -6695.214} C_VEL
LIN {X 0,Y 617.09,Z 251.696,A -85,B 0,C 180,E1 -6696.203,E2 -6696.203} C_VEL
LIN {X 0,Y 607.428,Z 226.45,A -85,B 0,C 180,E1 -6698.6,E2 -6698.6} C_VEL
LIN {X 0,Y 601.069,Z 210.359,A -85,B 0,C 180,E1 -6700.221,E2 -6700.221} C_VEL
LIN {X 0,Y 601.14,Z 210.349,A -85,B 0,C 180,E1 -6703.259,E2 -6703.259} C_VEL
LIN {X 0,Y 601.131,Z 210.351,A -85,B 0,C 180,E1 -6706.488,E2 -6706.488} C_VEL
LIN {X 0,Y 601.107,Z 210.401,A -85,B 0,C 180,E1 -6708.608,E2 -6708.608} C_VEL
LIN {X 0,Y 602.316,Z 213.709,A -85,B 0,C 180,E1 -6708.91,E2 -6708.91} C_VEL
LIN {X 0,Y 609.678,Z 230.052,A -85,B 0,C 180,E1 -6710.575,E2 -6710.575} C_VEL
LIN {X 0,Y 616.94,Z 248.368,A -85,B 0,C 180,E1 -6712.454,E2 -6712.454} C_VEL
LIN {X 0,Y 620.346,Z 257.325,A -85,B 0,C 180,E1 -6713.389,E2 -6713.389} C_VEL
LIN {X 0,Y 619.056,Z 301.971,A -85,B 0,C 180,E1 -6716.622,E2 -6716.622} C_VEL
LIN {X 0,Y 619.115,Z 330.54,A -85,B 0,C 180,E1 -6718.511,E2 -6718.511} C_VEL
LIN {X 0,Y 619.023,Z 333.002,A -85,B 0,C 180,E1 -6718.614,E2 -6718.614} C_VEL
LIN {X 0,Y 617.053,Z 436.465,A -85,B 0,C 180,E1 -6719.976,E2 -6719.976} C_VEL
LIN {X 0,Y 614.006,Z 548.9,A -85,B 0,C 180,E1 -6721.647,E2 -6721.647} C_VEL
LIN {X 0,Y 611.96,Z 623.565,A -85,B 0,C 180,E1 -6722.858,E2 -6722.858} C_VEL
LIN {X 0,Y 611.256,Z 645.434,A -85,B 0,C 180,E1 -6723.387,E2 -6723.387} C_VEL
LIN {X 0,Y 610.36,Z 666.913,A -85,B 0,C 180,E1 -6724.076,E2 -6724.076} C_VEL
LIN {X 0,Y 609.344,Z 688.042,A -85,B 0,C 180,E1 -6724.931,E2 -6724.931} C_VEL
LIN {X 0,Y 608.275,Z 707.568,A -85,B 0,C 180,E1 -6725.89,E2 -6725.89} C_VEL
LIN {X 0,Y 607.029,Z 728.422,A -85,B 0,C 180,E1 -6727.124,E2 -6727.124} C_VEL
LIN {X 0,Y 605.838,Z 747.388,A -85,B 0,C 180,E1 -6728.456,E2 -6728.456} C_VEL
LIN {X 0,Y 604.738,Z 764.055,A -85,B 0,C 180,E1 -6729.834,E2 -6729.834} C_VEL
LIN {X 0,Y 603.705,Z 779.814,A -85,B 0,C 180,E1 -6731.358,E2 -6731.358} C_VEL
LIN {X 0,Y 602.798,Z 793.738,A -85,B 0,C 180,E1 -6732.926,E2 -6732.926} C_VEL
LIN {X 0,Y 602.008,Z 806.213,A -85,B 0,C 180,E1 -6734.589,E2 -6734.589} C_VEL
LIN {X 0,Y 601.348,Z 817.34,A -85,B 0,C 180,E1 -6736.343,E2 -6736.343} C_VEL
LIN {X 0,Y 600.838,Z 827.201,A -85,B 0,C 180,E1 -6738.188,E2 -6738.188} C_VEL
LIN {X 0,Y 600.475,Z 835.217,A -85,B 0,C 180,E1 -6740.027,E2 -6740.027} C_VEL
LIN {X 0,Y 600.224,Z 842.262,A -85,B 0,C 180,E1 -6742.052,E2 -6742.052} C_VEL
LIN {X 0,Y 600.103,Z 847.613,A -85,B 0,C 180,E1 -6744.07,E2 -6744.07} C_VEL
LIN {X 0,Y 600.037,Z 851.301,A -85,B 0,C 180,E1 -6746.082,E2 -6746.082} C_VEL
LIN {X 0,Y 600.016,Z 853.513,A -85,B 0,C 180,E1 -6748.186,E2 -6748.186} C_VEL
LIN {X 0,Y 600.006,Z 854.165,A -85,B 0,C 180,E1 -6750.286,E2 -6750.286} C_VEL
LIN {X 0,Y 600.012,Z 853.186,A -85,B 0,C 180,E1 -6752.388,E2 -6752.388} C_VEL
LIN {X 0,Y 600.052,Z 850.676,A -85,B 0,C 180,E1 -6754.396,E2 -6754.396} C_VEL
LIN {X 0,Y 600.131,Z 846.465,A -85,B 0,C 180,E1 -6756.505,E2 -6756.505} C_VEL
LIN {X 0,Y 600.284,Z 840.789,A -85,B 0,C 180,E1 -6758.525,E2 -6758.525} C_VEL
LIN {X 0,Y 600.569,Z 833.231,A -85,B 0,C 180,E1 -6760.553,E2 -6760.553} C_VEL
LIN {X 0,Y 600.973,Z 824.228,A -85,B 0,C 180,E1 -6762.491,E2 -6762.491} C_VEL
LIN {X 0,Y 601.547,Z 813.84,A -85,B 0,C 180,E1 -6764.339,E2 -6764.339} C_VEL
LIN {X 0,Y 602.272,Z 801.989,A -85,B 0,C 180,E1 -6766.096,E2 -6766.096} C_VEL
LIN {X 0,Y 603.118,Z 788.653,A -85,B 0,C 180,E1 -6767.761,E2 -6767.761} C_VEL
LIN {X 0,Y 604.152,Z 772.909,A -85,B 0,C 180,E1 -6769.43,E2 -6769.43} C_VEL
LIN {X 0,Y 605.205,Z 757.135,A -85,B 0,C 180,E1 -6770.857,E2 -6770.857} C_VEL
LIN {X 0,Y 606.362,Z 739.202,A -85,B 0,C 180,E1 -6772.237,E2 -6772.237} C_VEL
LIN {X 0,Y 607.618,Z 718.665,A -85,B 0,C 180,E1 -6773.571,E2 -6773.571} C_VEL
LIN {X 0,Y 608.767,Z 698.662,A -85,B 0,C 180,E1 -6774.657,E2 -6774.657} C_VEL
LIN {X 0,Y 609.835,Z 678.194,A -85,B 0,C 180,E1 -6775.58,E2 -6775.58} C_VEL
LIN {X 0,Y 610.848,Z 655.983,A -85,B 0,C 180,E1 -6776.386,E2 -6776.386} C_VEL
LIN {X 0,Y 611.622,Z 634.616,A -85,B 0,C 180,E1 -6776.986,E2 -6776.986} C_VEL
LIN {X 0,Y 612.258,Z 612.134,A -85,B 0,C 180,E1 -6777.442,E2 -6777.442} C_VEL
LIN {X 0,Y 616.092,Z 474.409,A -85,B 0,C 180,E1 -6779.571,E2 -6779.571} C_VEL
LIN {X 0,Y 618.233,Z 380.383,A -85,B 0,C 180,E1 -6780.872,E2 -6780.872} C_VEL
LIN {X 0,Y 619.158,Z 331.734,A -85,B 0,C 180,E1 -6781.509,E2 -6781.509} C_VEL
LIN {X 0,Y 619.032,Z 304.277,A -85,B 0,C 180,E1 -6783.311,E2 -6783.311} C_VEL
LIN {X 0,Y 620.167,Z 264.814,A -85,B 0,C 180,E1 -6786.164,E2 -6786.164} C_VEL
LIN {X 0,Y 620.21,Z 257,A -85,B 0,C 180,E1 -6786.75,E2 -6786.75} C_VEL
LIN {X 0,Y 612.431,Z 236.635,A -85,B 0,C 180,E1 -6788.851,E2 -6788.851} C_VEL
LIN {X 0,Y 604.446,Z 218.015,A -85,B 0,C 180,E1 -6790.743,E2 -6790.743} C_VEL
LIN {X 0,Y 601.233,Z 211.02,A -85,B 0,C 180,E1 -6791.445,E2 -6791.445} C_VEL
LIN {X 0,Y 601.127,Z 210.345,A -85,B 0,C 180,E1 -6791.538,E2 -6791.538} C_VEL
LIN {X 0,Y 601.116,Z 210.356,A -85,B 0,C 180,E1 -6794.852,E2 -6794.852} C_VEL
LIN {X 0,Y 601.131,Z 210.356,A -85,B 0,C 180,E1 -6798.035,E2 -6798.035} C_VEL
LIN {X 0,Y 601.114,Z 210.353,A -85,B 0,C 180,E1 -6801.163,E2 -6801.163} C_VEL
LIN {X 0,Y 601.131,Z 210.349,A -85,B 0,C 180,E1 -6804.396,E2 -6804.396} C_VEL
LIN {X 0,Y 601.129,Z 210.338,A -85,B 0,C 180,E1 -6807.67,E2 -6807.67} C_VEL
LIN {X 0,Y 601.123,Z 210.341,A -85,B 0,C 180,E1 -6810.941,E2 -6810.941} C_VEL
LIN {X 0,Y 601.125,Z 210.349,A -85,B 0,C 180,E1 -6814.164,E2 -6814.164} C_VEL
LIN {X 0,Y 601.119,Z 210.333,A -85,B 0,C 180,E1 -6817.403,E2 -6817.403} C_VEL
LIN {X 0,Y 601.127,Z 210.338,A -85,B 0,C 180,E1 -6820.583,E2 -6820.583} C_VEL
LIN {X 0,Y 601.132,Z 210.346,A -85,B 0,C 180,E1 -6823.872,E2 -6823.872} C_VEL
LIN {X 0,Y 601.127,Z 210.333,A -85,B 0,C 180,E1 -6827.121,E2 -6827.121} C_VEL
LIN {X 0,Y 601.115,Z 210.351,A -85,B 0,C 180,E1 -6830.328,E2 -6830.328} C_VEL
LIN {X 0,Y 601.126,Z 210.33,A -85,B 0,C 180,E1 -6833.505,E2 -6833.505} C_VEL
LIN {X 0,Y 601.122,Z 210.347,A -85,B 0,C 180,E1 -6836.758,E2 -6836.758} C_VEL
LIN {X 0,Y 601.116,Z 210.326,A -85,B 0,C 180,E1 -6840.095,E2 -6840.095} C_VEL
LIN {X 0,Y 601.131,Z 210.347,A -85,B 0,C 180,E1 -6843.337,E2 -6843.337} C_VEL
LIN {X 0,Y 601.104,Z 210.328,A -85,B 0,C 180,E1 -6846.495,E2 -6846.495} C_VEL
LIN {X 0,Y 601.133,Z 210.347,A -85,B 0,C 180,E1 -6849.671,E2 -6849.671} C_VEL
LIN {X 0,Y 601.117,Z 210.347,A -85,B 0,C 180,E1 -6852.904,E2 -6852.904} C_VEL
LIN {X 0,Y 601.107,Z 210.355,A -85,B 0,C 180,E1 -6856.228,E2 -6856.228} C_VEL
LIN {X 0,Y 601.137,Z 210.346,A -85,B 0,C 180,E1 -6859.431,E2 -6859.431} C_VEL
LIN {X 0,Y 601.097,Z 210.354,A -85,B 0,C 180,E1 -6862.6,E2 -6862.6} C_VEL
LIN {X 0,Y 601.137,Z 210.354,A -85,B 0,C 180,E1 -6865.73,E2 -6865.73} C_VEL
LIN {X 0,Y 601.099,Z 210.35,A -85,B 0,C 180,E1 -6868.842,E2 -6868.842} C_VEL
LIN {X 0,Y 601.122,Z 210.35,A -85,B 0,C 180,E1 -6872.047,E2 -6872.047} C_VEL
LIN {X 0,Y 601.11,Z 210.352,A -85,B 0,C 180,E1 -6875.138,E2 -6875.138} C_VEL
LIN {X 0,Y 601.093,Z 210.352,A -85,B 0,C 180,E1 -6878.419,E2 -6878.419} C_VEL
LIN {X 0,Y 601.149,Z 210.526,A -85,B 0,C 180,E1 -6881.359,E2 -6881.359} C_VEL
LIN {X 0,Y 602.474,Z 213.87,A -85,B 0,C 180,E1 -6881.722,E2 -6881.722} C_VEL
LIN {X 0,Y 603.677,Z 216.239,A -85,B 0,C 180,E1 -6882.002,E2 -6882.002} C_VEL
LIN {X 0,Y 612.281,Z 233.182,A -85,B 0,C 180,E1 -6883.952,E2 -6883.952} C_VEL
LIN {X 0,Y 623.73,Z 256.375,A -85,B 0,C 180,E1 -6886.423,E2 -6886.423} C_VEL
LIN {X 0,Y 627.625,Z 264.84,A -85,B 0,C 180,E1 -6887.26,E2 -6887.26} C_VEL
LIN {X 0,Y 624.68,Z 306.779,A -85,B 0,C 180,E1 -6889.509,E2 -6889.509} C_VEL
LIN {X 0,Y 627.288,Z 327.204,A -85,B 0,C 180,E1 -6889.995,E2 -6889.995} C_VEL
LIN {X 0,Y 622.673,Z 577.422,A -85,B 0,C 180,E1 -6893.305,E2 -6893.305} C_VEL
LIN {X 0,Y 620.808,Z 692.639,A -85,B 0,C 180,E1 -6894.795,E2 -6894.795} C_VEL
LIN {X 0,Y 619.891,Z 717.552,A -85,B 0,C 180,E1 -6895.278,E2 -6895.278} C_VEL
LIN {X 0,Y 618.86,Z 738.778,A -85,B 0,C 180,E1 -6895.824,E2 -6895.824} C_VEL
LIN {X 0,Y 617.374,Z 764.189,A -85,B 0,C 180,E1 -6896.658,E2 -6896.658} C_VEL
LIN {X 0,Y 615.935,Z 785.11,A -85,B 0,C 180,E1 -6897.498,E2 -6897.498} C_VEL
LIN {X 0,Y 614.215,Z 808.946,A -85,B 0,C 180,E1 -6898.644,E2 -6898.644} C_VEL
LIN {X 0,Y 612.615,Z 828.882,A -85,B 0,C 180,E1 -6899.767,E2 -6899.767} C_VEL
LIN {X 0,Y 610.668,Z 851.586,A -85,B 0,C 180,E1 -6901.251,E2 -6901.251} C_VEL
LIN {X 0,Y 609.029,Z 870.543,A -85,B 0,C 180,E1 -6902.68,E2 -6902.68} C_VEL
LIN {X 0,Y 607.278,Z 890.328,A -85,B 0,C 180,E1 -6904.392,E2 -6904.392} C_VEL
LIN {X 0,Y 605.874,Z 906.64,A -85,B 0,C 180,E1 -6905.996,E2 -6905.996} C_VEL
LIN {X 0,Y 604.409,Z 923.986,A -85,B 0,C 180,E1 -6907.943,E2 -6907.943} C_VEL
LIN {X 0,Y 603.355,Z 935.91,A -85,B 0,C 180,E1 -6909.533,E2 -6909.533} C_VEL
LIN {X 0,Y 602.248,Z 949.662,A -85,B 0,C 180,E1 -6911.612,E2 -6911.612} C_VEL
LIN {X 0,Y 601.41,Z 961.308,A -85,B 0,C 180,E1 -6913.682,E2 -6913.682} C_VEL
LIN {X 0,Y 600.821,Z 971.391,A -85,B 0,C 180,E1 -6915.741,E2 -6915.741} C_VEL
LIN {X 0,Y 600.388,Z 980.543,A -85,B 0,C 180,E1 -6917.985,E2 -6917.985} C_VEL
LIN {X 0,Y 600.133,Z 987.422,A -85,B 0,C 180,E1 -6920.022,E2 -6920.022} C_VEL
LIN {X 0,Y 599.961,Z 993.863,A -85,B 0,C 180,E1 -6922.434,E2 -6922.434} C_VEL
LIN {X 0,Y 599.914,Z 997.814,A -85,B 0,C 180,E1 -6924.453,E2 -6924.453} C_VEL
LIN {X 0,Y 599.907,Z 1000.69,A -85,B 0,C 180,E1 -6926.56,E2 -6926.56} C_VEL
LIN {X 0,Y 599.902,Z 1002.258,A -85,B 0,C 180,E1 -6928.95,E2 -6928.95} C_VEL
LIN {X 0,Y 599.89,Z 1002.304,A -85,B 0,C 180,E1 -6930.86,E2 -6930.86} C_VEL
LIN {X 0,Y 599.888,Z 1001.086,A -85,B 0,C 180,E1 -6933.058,E2 -6933.058} C_VEL
LIN {X 0,Y 599.905,Z 998.132,A -85,B 0,C 180,E1 -6935.356,E2 -6935.356} C_VEL
LIN {X 0,Y 599.962,Z 994.482,A -85,B 0,C 180,E1 -6937.277,E2 -6937.277} C_VEL
LIN {X 0,Y 600.113,Z 988.633,A -85,B 0,C 180,E1 -6939.591,E2 -6939.591} C_VEL
LIN {X 0,Y 600.332,Z 981.6,A -85,B 0,C 180,E1 -6941.724,E2 -6941.724} C_VEL
LIN {X 0,Y 600.696,Z 973.533,A -85,B 0,C 180,E1 -6943.77,E2 -6943.77} C_VEL
LIN {X 0,Y 601.309,Z 962.843,A -85,B 0,C 180,E1 -6946.026,E2 -6946.026} C_VEL
LIN {X 0,Y 602.029,Z 952.538,A -85,B 0,C 180,E1 -6947.894,E2 -6947.894} C_VEL
LIN {X 0,Y 603.139,Z 938.712,A -85,B 0,C 180,E1 -6950.07,E2 -6950.07} C_VEL
LIN {X 0,Y 604.242,Z 925.857,A -85,B 0,C 180,E1 -6951.823,E2 -6951.823} C_VEL
LIN {X 0,Y 605.106,Z 915.265,A -85,B 0,C 180,E1 -6953.056,E2 -6953.056} C_VEL
LIN {X 0,Y 606.516,Z 898.257,A -85,B 0,C 180,E1 -6954.807,E2 -6954.807} C_VEL
LIN {X 0,Y 608.005,Z 879.617,A -85,B 0,C 180,E1 -6956.466,E2 -6956.466} C_VEL
LIN {X 0,Y 609.641,Z 859.612,A -85,B 0,C 180,E1 -6958.032,E2 -6958.032} C_VEL
LIN {X 0,Y 611.205,Z 838.818,A -85,B 0,C 180,E1 -6959.428,E2 -6959.428} C_VEL
LIN {X 0,Y 612.789,Z 816.849,A -85,B 0,C 180,E1 -6960.712,E2 -6960.712} C_VEL
LIN {X 0,Y 614.229,Z 795.108,A -85,B 0,C 180,E1 -6961.783,E2 -6961.783} C_VEL
LIN {X 0,Y 615.576,Z 772.242,A -85,B 0,C 180,E1 -6962.745,E2 -6962.745} C_VEL
LIN {X 0,Y 616.728,Z 749.003,A -85,B 0,C 180,E1 -6963.536,E2 -6963.536} C_VEL
LIN {X 0,Y 617.781,Z 724.379,A -85,B 0,C 180,E1 -6964.208,E2 -6964.208} C_VEL
LIN {X 0,Y 618.516,Z 701.498,A -85,B 0,C 180,E1 -6964.672,E2 -6964.672} C_VEL
LIN {X 0,Y 619.007,Z 675.507,A -85,B 0,C 180,E1 -6965.043,E2 -6965.043} C_VEL
LIN {X 0,Y 620.538,Z 501.987,A -85,B 0,C 180,E1 -6967.118,E2 -6967.118} C_VEL
LIN {X 0,Y 622.659,Z 358.927,A -85,B 0,C 180,E1 -6968.99,E2 -6968.99} C_VEL
LIN {X 0,Y 623.157,Z 323.924,A -85,B 0,C 180,E1 -6969.489,E2 -6969.489} C_VEL
LIN {X 0,Y 622.423,Z 317.936,A -85,B 0,C 180,E1 -6969.655,E2 -6969.655} C_VEL
LIN {X 0,Y 625.911,Z 290.989,A -85,B 0,C 180,E1 -6971.338,E2 -6971.338} C_VEL
LIN {X 0,Y 630.454,Z 267.29,A -85,B 0,C 180,E1 -6972.967,E2 -6972.967} C_VEL
LIN {X 0,Y 628.203,Z 260.386,A -85,B 0,C 180,E1 -6974.123,E2 -6974.123} C_VEL
LIN {X 0,Y 626.415,Z 255.361,A -85,B 0,C 180,E1 -6975.261,E2 -6975.261} C_VEL
LIN {X 0,Y 625.348,Z 252.472,A -85,B 0,C 180,E1 -6976.184,E2 -6976.184} C_VEL
LIN {X 0,Y 624.567,Z 249.826,A -85,B 0,C 180,E1 -6977.7,E2 -6977.7} C_VEL
LIN {X 0,Y 624.544,Z 249.642,A -85,B 0,C 180,E1 -6978.527,E2 -6978.527} C_VEL
LIN {X 0,Y 624.752,Z 251.749,A -85,B 0,C 180,E1 -6979.909,E2 -6979.909} C_VEL
LIN {X 0,Y 625.212,Z 253.057,A -85,B 0,C 180,E1 -6980.467,E2 -6980.467} C_VEL
LIN {X 0,Y 626.209,Z 256.598,A -85,B 0,C 180,E1 -6981.484,E2 -6981.484} C_VEL
LIN {X 0,Y 627.862,Z 262.844,A -85,B 0,C 180,E1 -6982.759,E2 -6982.759} C_VEL
LIN {X 0,Y 628.158,Z 264.412,A -85,B 0,C 180,E1 -6983.009,E2 -6983.009} C_VEL
LIN {X 0,Y 623.023,Z 289.132,A -85,B 0,C 180,E1 -6985.044,E2 -6985.044} C_VEL
LIN {X 0,Y 618.197,Z 322.726,A -85,B 0,C 180,E1 -6987.597,E2 -6987.597} C_VEL
LIN {X 0,Y 614.216,Z 363.397,A -85,B 0,C 180,E1 -6990.499,E2 -6990.499} C_VEL
LIN {X 0,Y 610.89,Z 409.635,A -85,B 0,C 180,E1 -6993.616,E2 -6993.616} C_VEL
LIN {X 0,Y 609.712,Z 432.322,A -85,B 0,C 180,E1 -6995.079,E2 -6995.079} C_VEL
LIN {X 0,Y 613.59,Z 467.49,A -85,B 0,C 180,E1 -6996.166,E2 -6996.166} C_VEL
LIN {X 0,Y 615.47,Z 490.857,A -85,B 0,C 180,E1 -6996.795,E2 -6996.795} C_VEL
LIN {X 0,Y 610.773,Z 599.976,A -85,B 0,C 180,E1 -6998.711,E2 -6998.711} C_VEL
LIN {X 0,Y 608.163,Z 686.24,A -85,B 0,C 180,E1 -7000.162,E2 -7000.162} C_VEL
LIN {X 0,Y 607.423,Z 708.178,A -85,B 0,C 180,E1 -7000.719,E2 -7000.719} C_VEL
LIN {X 0,Y 606.694,Z 727.93,A -85,B 0,C 180,E1 -7001.398,E2 -7001.398} C_VEL
LIN {X 0,Y 605.914,Z 746.818,A -85,B 0,C 180,E1 -7002.224,E2 -7002.224} C_VEL
LIN {X 0,Y 605.16,Z 764.688,A -85,B 0,C 180,E1 -7003.193,E2 -7003.193} C_VEL
LIN {X 0,Y 604.392,Z 781.505,A -85,B 0,C 180,E1 -7004.307,E2 -7004.307} C_VEL
LIN {X 0,Y 603.636,Z 797.159,A -85,B 0,C 180,E1 -7005.564,E2 -7005.564} C_VEL
LIN {X 0,Y 602.971,Z 810.645,A -85,B 0,C 180,E1 -7006.869,E2 -7006.869} C_VEL
LIN {X 0,Y 602.351,Z 823.282,A -85,B 0,C 180,E1 -7008.347,E2 -7008.347} C_VEL
LIN {X 0,Y 601.837,Z 833.841,A -85,B 0,C 180,E1 -7009.857,E2 -7009.857} C_VEL
LIN {X 0,Y 601.404,Z 843.037,A -85,B 0,C 180,E1 -7011.491,E2 -7011.491} C_VEL
LIN {X 0,Y 601.1,Z 850.268,A -85,B 0,C 180,E1 -7013.121,E2 -7013.121} C_VEL
LIN {X 0,Y 600.881,Z 855.972,A -85,B 0,C 180,E1 -7014.845,E2 -7014.845} C_VEL
LIN {X 0,Y 600.72,Z 859.869,A -85,B 0,C 180,E1 -7016.565,E2 -7016.565} C_VEL
LIN {X 0,Y 600.611,Z 862.12,A -85,B 0,C 180,E1 -7018.378,E2 -7018.378} C_VEL
LIN {X 0,Y 600.559,Z 862.545,A -85,B 0,C 180,E1 -7020.191,E2 -7020.191} C_VEL
LIN {X 0,Y 600.538,Z 861.171,A -85,B 0,C 180,E1 -7022.004,E2 -7022.004} C_VEL
LIN {X 0,Y 600.564,Z 858.217,A -85,B 0,C 180,E1 -7023.723,E2 -7023.723} C_VEL
LIN {X 0,Y 600.657,Z 853.536,A -85,B 0,C 180,E1 -7025.456,E2 -7025.456} C_VEL
LIN {X 0,Y 600.806,Z 847.121,A -85,B 0,C 180,E1 -7027.17,E2 -7027.17} C_VEL
LIN {X 0,Y 601.056,Z 839.076,A -85,B 0,C 180,E1 -7028.828,E2 -7028.828} C_VEL
LIN {X 0,Y 601.429,Z 829.289,A -85,B 0,C 180,E1 -7030.441,E2 -7030.441} C_VEL
LIN {X 0,Y 601.919,Z 817.817,A -85,B 0,C 180,E1 -7031.985,E2 -7031.985} C_VEL
LIN {X 0,Y 602.52,Z 804.779,A -85,B 0,C 180,E1 -7033.434,E2 -7033.434} C_VEL
LIN {X 0,Y 603.222,Z 790.109,A -85,B 0,C 180,E1 -7034.79,E2 -7034.79} C_VEL
LIN {X 0,Y 603.983,Z 774.321,A -85,B 0,C 180,E1 -7036,E2 -7036} C_VEL
LIN {X 0,Y 604.744,Z 757.506,A -85,B 0,C 180,E1 -7037.067,E2 -7037.067} C_VEL
LIN {X 0,Y 605.528,Z 739.712,A -85,B 0,C 180,E1 -7037.986,E2 -7037.986} C_VEL
LIN {X 0,Y 606.282,Z 720.913,A -85,B 0,C 180,E1 -7038.76,E2 -7038.76} C_VEL
LIN {X 0,Y 606.939,Z 701.311,A -85,B 0,C 180,E1 -7039.375,E2 -7039.375} C_VEL
LIN {X 0,Y 607.504,Z 680.839,A -85,B 0,C 180,E1 -7039.828,E2 -7039.828} C_VEL
LIN {X 0,Y 610.916,Z 486.571,A -85,B 0,C 180,E1 -7042.555,E2 -7042.555} C_VEL
LIN {X 0,Y 607.601,Z 458.258,A -85,B 0,C 180,E1 -7043.132,E2 -7043.132} C_VEL
LIN {X 0,Y 609.616,Z 407.306,A -85,B 0,C 180,E1 -7046.286,E2 -7046.286} C_VEL
LIN {X 0,Y 611.998,Z 354.957,A -85,B 0,C 180,E1 -7049.565,E2 -7049.565} C_VEL
LIN {X 0,Y 613.838,Z 316.525,A -85,B 0,C 180,E1 -7052.005,E2 -7052.005} C_VEL
LIN {X 0,Y 613.281,Z 310.388,A -85,B 0,C 180,E1 -7052.445,E2 -7052.445} C_VEL
LIN {X 0,Y 608.553,Z 295.028,A -85,B 0,C 180,E1 -7053.751,E2 -7053.751} C_VEL
LIN {X 0,Y 608.182,Z 289.748,A -85,B 0,C 180,E1 -7054.133,E2 -7054.133} C_VEL
LIN {X 0,Y 610.078,Z 254.976,A -85,B 0,C 180,E1 -7056.416,E2 -7056.416} C_VEL
LIN {X 0,Y 600.345,Z 229.525,A -85,B 0,C 180,E1 -7058.864,E2 -7058.864} C_VEL
LIN {X 0,Y 593.135,Z 211.351,A -85,B 0,C 180,E1 -7060.723,E2 -7060.723} C_VEL
LIN {X 0,Y 593.169,Z 211.344,A -85,B 0,C 180,E1 -7063.988,E2 -7063.988} C_VEL
LIN {X 0,Y 593.18,Z 211.337,A -85,B 0,C 180,E1 -7067.16,E2 -7067.16} C_VEL
LIN {X 0,Y 593.218,Z 211.467,A -85,B 0,C 180,E1 -7068.027,E2 -7068.027} C_VEL
LIN {X 0,Y 594.379,Z 214.664,A -85,B 0,C 180,E1 -7068.324,E2 -7068.324} C_VEL
LIN {X 0,Y 600.487,Z 227.959,A -85,B 0,C 180,E1 -7069.697,E2 -7069.697} C_VEL
LIN {X 0,Y 607.068,Z 243.692,A -85,B 0,C 180,E1 -7071.327,E2 -7071.327} C_VEL
LIN {X 0,Y 613.657,Z 261.319,A -85,B 0,C 180,E1 -7073.157,E2 -7073.157} C_VEL
LIN {X 0,Y 612.425,Z 305.402,A -85,B 0,C 180,E1 -7076.338,E2 -7076.338} C_VEL
LIN {X 0,Y 612.539,Z 333.426,A -85,B 0,C 180,E1 -7078.18,E2 -7078.18} C_VEL
LIN {X 0,Y 612.203,Z 336.182,A -85,B 0,C 180,E1 -7078.255,E2 -7078.255} C_VEL
LIN {X 0,Y 610.183,Z 437.088,A -85,B 0,C 180,E1 -7079.598,E2 -7079.598} C_VEL
LIN {X 0,Y 607.137,Z 543.148,A -85,B 0,C 180,E1 -7081.198,E2 -7081.198} C_VEL
LIN {X 0,Y 604.719,Z 624.048,A -85,B 0,C 180,E1 -7082.541,E2 -7082.541} C_VEL
LIN {X 0,Y 603.991,Z 645.916,A -85,B 0,C 180,E1 -7083.074,E2 -7083.074} C_VEL
LIN {X 0,Y 603.024,Z 668.157,A -85,B 0,C 180,E1 -7083.796,E2 -7083.796} C_VEL
LIN {X 0,Y 601.937,Z 689.333,A -85,B 0,C 180,E1 -7084.67,E2 -7084.67} C_VEL
LIN {X 0,Y 600.766,Z 709.275,A -85,B 0,C 180,E1 -7085.674,E2 -7085.674} C_VEL
LIN {X 0,Y 599.435,Z 729.797,A -85,B 0,C 180,E1 -7086.921,E2 -7086.921} C_VEL
LIN {X 0,Y 598.109,Z 749.038,A -85,B 0,C 180,E1 -7088.318,E2 -7088.318} C_VEL
LIN {X 0,Y 596.935,Z 765.546,A -85,B 0,C 180,E1 -7089.723,E2 -7089.723} C_VEL
LIN {X 0,Y 595.841,Z 781.606,A -85,B 0,C 180,E1 -7091.306,E2 -7091.306} C_VEL
LIN {X 0,Y 594.911,Z 795.43,A -85,B 0,C 180,E1 -7092.895,E2 -7092.895} C_VEL
LIN {X 0,Y 594.069,Z 808.584,A -85,B 0,C 180,E1 -7094.678,E2 -7094.678} C_VEL
LIN {X 0,Y 593.393,Z 819.658,A -85,B 0,C 180,E1 -7096.476,E2 -7096.476} C_VEL
LIN {X 0,Y 592.86,Z 829.665,A -85,B 0,C 180,E1 -7098.422,E2 -7098.422} C_VEL
LIN {X 0,Y 592.523,Z 837.529,A -85,B 0,C 180,E1 -7100.285,E2 -7100.285} C_VEL
LIN {X 0,Y 592.279,Z 844.168,A -85,B 0,C 180,E1 -7102.3,E2 -7102.3} C_VEL
LIN {X 0,Y 592.15,Z 849.317,A -85,B 0,C 180,E1 -7104.38,E2 -7104.38} C_VEL
LIN {X 0,Y 592.102,Z 852.82,A -85,B 0,C 180,E1 -7106.418,E2 -7106.418} C_VEL
LIN {X 0,Y 592.07,Z 854.699,A -85,B 0,C 180,E1 -7108.452,E2 -7108.452} C_VEL
LIN {X 0,Y 592.058,Z 855.094,A -85,B 0,C 180,E1 -7110.581,E2 -7110.581} C_VEL
LIN {X 0,Y 592.081,Z 854.009,A -85,B 0,C 180,E1 -7112.613,E2 -7112.613} C_VEL
LIN {X 0,Y 592.127,Z 851.322,A -85,B 0,C 180,E1 -7114.649,E2 -7114.649} C_VEL
LIN {X 0,Y 592.203,Z 846.867,A -85,B 0,C 180,E1 -7116.788,E2 -7116.788} C_VEL
LIN {X 0,Y 592.383,Z 840.937,A -85,B 0,C 180,E1 -7118.836,E2 -7118.836} C_VEL
LIN {X 0,Y 592.704,Z 833.557,A -85,B 0,C 180,E1 -7120.793,E2 -7120.793} C_VEL
LIN {X 0,Y 593.108,Z 824.814,A -85,B 0,C 180,E1 -7122.66,E2 -7122.66} C_VEL
LIN {X 0,Y 593.707,Z 814.242,A -85,B 0,C 180,E1 -7124.533,E2 -7124.533} C_VEL
LIN {X 0,Y 594.473,Z 802.239,A -85,B 0,C 180,E1 -7126.313,E2 -7126.313} C_VEL
LIN {X 0,Y 595.364,Z 788.692,A -85,B 0,C 180,E1 -7128,E2 -7128} C_VEL
LIN {X 0,Y 596.373,Z 773.725,A -85,B 0,C 180,E1 -7129.592,E2 -7129.592} C_VEL
LIN {X 0,Y 597.545,Z 756.864,A -85,B 0,C 180,E1 -7131.13,E2 -7131.13} C_VEL
LIN {X 0,Y 598.763,Z 739.646,A -85,B 0,C 180,E1 -7132.483,E2 -7132.483} C_VEL
LIN {X 0,Y 600.067,Z 720.184,A -85,B 0,C 180,E1 -7133.781,E2 -7133.781} C_VEL
LIN {X 0,Y 601.29,Z 700.488,A -85,B 0,C 180,E1 -7134.88,E2 -7134.88} C_VEL
LIN {X 0,Y 602.434,Z 679.975,A -85,B 0,C 180,E1 -7135.829,E2 -7135.829} C_VEL
LIN {X 0,Y 603.507,Z 657.848,A -85,B 0,C 180,E1 -7136.652,E2 -7136.652} C_VEL
LIN {X 0,Y 604.338,Z 636.285,A -85,B 0,C 180,E1 -7137.274,E2 -7137.274} C_VEL
LIN {X 0,Y 605.009,Z 613.854,A -85,B 0,C 180,E1 -7137.742,E2 -7137.742} C_VEL
LIN {X 0,Y 608.853,Z 486.088,A -85,B 0,C 180,E1 -7139.775,E2 -7139.775} C_VEL
LIN {X 0,Y 611.155,Z 394.563,A -85,B 0,C 180,E1 -7141.078,E2 -7141.078} C_VEL
LIN {X 0,Y 612.283,Z 334.674,A -85,B 0,C 180,E1 -7141.863,E2 -7141.863} C_VEL
LIN {X 0,Y 612.54,Z 332.282,A -85,B 0,C 180,E1 -7141.985,E2 -7141.985} C_VEL
LIN {X 0,Y 612.47,Z 304.376,A -85,B 0,C 180,E1 -7143.828,E2 -7143.828} C_VEL
LIN {X 0,Y 613.671,Z 261.933,A -85,B 0,C 180,E1 -7146.894,E2 -7146.894} C_VEL
LIN {X 0,Y 612.969,Z 259.122,A -85,B 0,C 180,E1 -7147.161,E2 -7147.161} C_VEL
LIN {X 0,Y 604.957,Z 238.295,A -85,B 0,C 180,E1 -7149.328,E2 -7149.328} C_VEL
LIN {X 0,Y 597.566,Z 221.41,A -85,B 0,C 180,E1 -7151.078,E2 -7151.078} C_VEL
LIN {X 0,Y 594.239,Z 214.4,A -85,B 0,C 180,E1 -7151.805,E2 -7151.805} C_VEL
LIN {X 0,Y 593.193,Z 211.342,A -85,B 0,C 180,E1 -7152.095,E2 -7152.095} C_VEL
LIN {X 0,Y 593.178,Z 211.346,A -85,B 0,C 180,E1 -7155.344,E2 -7155.344} C_VEL
LIN {X 0,Y 593.193,Z 211.34,A -85,B 0,C 180,E1 -7158.642,E2 -7158.642} C_VEL
LIN {X 0,Y 593.193,Z 211.337,A -85,B 0,C 180,E1 -7161.923,E2 -7161.923} C_VEL
LIN {X 0,Y 593.177,Z 211.341,A -85,B 0,C 180,E1 -7165.176,E2 -7165.176} C_VEL
LIN {X 0,Y 593.192,Z 211.337,A -85,B 0,C 180,E1 -7168.384,E2 -7168.384} C_VEL
LIN {X 0,Y 593.194,Z 211.322,A -85,B 0,C 180,E1 -7171.629,E2 -7171.629} C_VEL
LIN {X 0,Y 593.186,Z 211.335,A -85,B 0,C 180,E1 -7174.97,E2 -7174.97} C_VEL
LIN {X 0,Y 593.184,Z 211.337,A -85,B 0,C 180,E1 -7178.128,E2 -7178.128} C_VEL
LIN {X 0,Y 593.184,Z 211.321,A -85,B 0,C 180,E1 -7181.321,E2 -7181.321} C_VEL
LIN {X 0,Y 593.185,Z 211.335,A -85,B 0,C 180,E1 -7184.554,E2 -7184.554} C_VEL
LIN {X 0,Y 593.188,Z 211.315,A -85,B 0,C 180,E1 -7187.867,E2 -7187.867} C_VEL
LIN {X 0,Y 593.19,Z 211.337,A -85,B 0,C 180,E1 -7191.176,E2 -7191.176} C_VEL
LIN {X 0,Y 593.172,Z 211.317,A -85,B 0,C 180,E1 -7194.292,E2 -7194.292} C_VEL
LIN {X 0,Y 593.191,Z 211.34,A -85,B 0,C 180,E1 -7197.488,E2 -7197.488} C_VEL
LIN {X 0,Y 593.174,Z 211.311,A -85,B 0,C 180,E1 -7200.676,E2 -7200.676} C_VEL
LIN {X 0,Y 593.186,Z 211.343,A -85,B 0,C 180,E1 -7203.963,E2 -7203.963} C_VEL
LIN {X 0,Y 593.195,Z 211.309,A -85,B 0,C 180,E1 -7207.263,E2 -7207.263} C_VEL
LIN {X 0,Y 593.165,Z 211.34,A -85,B 0,C 180,E1 -7210.489,E2 -7210.489} C_VEL
LIN {X 0,Y 593.199,Z 211.342,A -85,B 0,C 180,E1 -7213.749,E2 -7213.749} C_VEL
LIN {X 0,Y 593.177,Z 211.339,A -85,B 0,C 180,E1 -7216.955,E2 -7216.955} C_VEL
LIN {X 0,Y 593.17,Z 211.342,A -85,B 0,C 180,E1 -7220.216,E2 -7220.216} C_VEL
LIN {X 0,Y 593.201,Z 211.34,A -85,B 0,C 180,E1 -7223.441,E2 -7223.441} C_VEL
LIN {X 0,Y 593.156,Z 211.336,A -85,B 0,C 180,E1 -7226.641,E2 -7226.641} C_VEL
LIN {X 0,Y 593.204,Z 211.336,A -85,B 0,C 180,E1 -7229.818,E2 -7229.818} C_VEL
LIN {X 0,Y 593.162,Z 211.342,A -85,B 0,C 180,E1 -7232.989,E2 -7232.989} C_VEL
LIN {X 0,Y 593.161,Z 211.34,A -85,B 0,C 180,E1 -7236.316,E2 -7236.316} C_VEL
LIN {X 0,Y 593.197,Z 211.336,A -85,B 0,C 180,E1 -7239.466,E2 -7239.466} C_VEL
LIN {X 0,Y 593.157,Z 211.411,A -85,B 0,C 180,E1 -7240.634,E2 -7240.634} C_VEL
LIN {X 0,Y 594.407,Z 214.747,A -85,B 0,C 180,E1 -7240.999,E2 -7240.999} C_VEL
LIN {X 0,Y 595.655,Z 216.909,A -85,B 0,C 180,E1 -7241.278,E2 -7241.278} C_VEL
LIN {X 0,Y 606.616,Z 238.67,A -85,B 0,C 180,E1 -7243.812,E2 -7243.812} C_VEL
LIN {X 0,Y 617.643,Z 261.089,A -85,B 0,C 180,E1 -7246.222,E2 -7246.222} C_VEL
LIN {X 0,Y 621.018,Z 268.672,A -85,B 0,C 180,E1 -7246.969,E2 -7246.969} C_VEL
LIN {X 0,Y 618.145,Z 307.382,A -85,B 0,C 180,E1 -7249.066,E2 -7249.066} C_VEL
LIN {X 0,Y 620.802,Z 328.6,A -85,B 0,C 180,E1 -7249.578,E2 -7249.578} C_VEL
LIN {X 0,Y 615.932,Z 572.75,A -85,B 0,C 180,E1 -7252.855,E2 -7252.855} C_VEL
LIN {X 0,Y 613.838,Z 692.54,A -85,B 0,C 180,E1 -7254.426,E2 -7254.426} C_VEL
LIN {X 0,Y 612.884,Z 717.171,A -85,B 0,C 180,E1 -7254.909,E2 -7254.909} C_VEL
LIN {X 0,Y 611.809,Z 738.227,A -85,B 0,C 180,E1 -7255.455,E2 -7255.455} C_VEL
LIN {X 0,Y 610.287,Z 763.159,A -85,B 0,C 180,E1 -7256.276,E2 -7256.276} C_VEL
LIN {X 0,Y 608.767,Z 784.121,A -85,B 0,C 180,E1 -7257.123,E2 -7257.123} C_VEL
LIN {X 0,Y 606.916,Z 808.338,A -85,B 0,C 180,E1 -7258.295,E2 -7258.295} C_VEL
LIN {X 0,Y 605.256,Z 828.024,A -85,B 0,C 180,E1 -7259.415,E2 -7259.415} C_VEL
LIN {X 0,Y 603.26,Z 850.119,A -85,B 0,C 180,E1 -7260.867,E2 -7260.867} C_VEL
LIN {X 0,Y 601.512,Z 869.179,A -85,B 0,C 180,E1 -7262.315,E2 -7262.315} C_VEL
LIN {X 0,Y 599.633,Z 889.578,A -85,B 0,C 180,E1 -7264.095,E2 -7264.095} C_VEL
LIN {X 0,Y 598.139,Z 905.898,A -85,B 0,C 180,E1 -7265.718,E2 -7265.718} C_VEL
LIN {X 0,Y 596.572,Z 923.686,A -85,B 0,C 180,E1 -7267.741,E2 -7267.741} C_VEL
LIN {X 0,Y 595.456,Z 936.908,A -85,B 0,C 180,E1 -7269.454,E2 -7269.454} C_VEL
LIN {X 0,Y 594.599,Z 947.776,A -85,B 0,C 180,E1 -7271.062,E2 -7271.062} C_VEL
LIN {X 0,Y 593.618,Z 960.277,A -85,B 0,C 180,E1 -7273.26,E2 -7273.26} C_VEL
LIN {X 0,Y 592.984,Z 970.014,A -85,B 0,C 180,E1 -7275.249,E2 -7275.249} C_VEL
LIN {X 0,Y 592.448,Z 980.189,A -85,B 0,C 180,E1 -7277.722,E2 -7277.722} C_VEL
LIN {X 0,Y 592.166,Z 987.119,A -85,B 0,C 180,E1 -7279.788,E2 -7279.788} C_VEL
LIN {X 0,Y 591.983,Z 993.449,A -85,B 0,C 180,E1 -7282.137,E2 -7282.137} C_VEL
LIN {X 0,Y 591.93,Z 997.654,A -85,B 0,C 180,E1 -7284.28,E2 -7284.28} C_VEL
LIN {X 0,Y 591.914,Z 1000.463,A -85,B 0,C 180,E1 -7286.32,E2 -7286.32} C_VEL
LIN {X 0,Y 591.908,Z 1002.213,A -85,B 0,C 180,E1 -7288.742,E2 -7288.742} C_VEL
LIN {X 0,Y 591.887,Z 1002.326,A -85,B 0,C 180,E1 -7290.774,E2 -7290.774} C_VEL
LIN {X 0,Y 591.886,Z 1001.29,A -85,B 0,C 180,E1 -7292.808,E2 -7292.808} C_VEL
LIN {X 0,Y 591.903,Z 998.451,A -85,B 0,C 180,E1 -7295.234,E2 -7295.234} C_VEL
LIN {X 0,Y 591.965,Z 994.688,A -85,B 0,C 180,E1 -7297.278,E2 -7297.278} C_VEL
LIN {X 0,Y 592.116,Z 989.184,A -85,B 0,C 180,E1 -7299.533,E2 -7299.533} C_VEL
LIN {X 0,Y 592.358,Z 981.952,A -85,B 0,C 180,E1 -7301.785,E2 -7301.785} C_VEL
LIN {X 0,Y 592.718,Z 974.342,A -85,B 0,C 180,E1 -7303.76,E2 -7303.76} C_VEL
LIN {X 0,Y 593.403,Z 963.252,A -85,B 0,C 180,E1 -7306.165,E2 -7306.165} C_VEL
LIN {X 0,Y 594.197,Z 952.536,A -85,B 0,C 180,E1 -7308.138,E2 -7308.138} C_VEL
LIN {X 0,Y 595.198,Z 940.599,A -85,B 0,C 180,E1 -7310.042,E2 -7310.042} C_VEL
LIN {X 0,Y 596.362,Z 925.486,A -85,B 0,C 180,E1 -7311.999,E2 -7311.999} C_VEL
LIN {X 0,Y 597.672,Z 909.919,A -85,B 0,C 180,E1 -7313.778,E2 -7313.778} C_VEL
LIN {X 0,Y 599.159,Z 891.995,A -85,B 0,C 180,E1 -7315.556,E2 -7315.556} C_VEL
LIN {X 0,Y 600.714,Z 873.905,A -85,B 0,C 180,E1 -7317.134,E2 -7317.134} C_VEL
LIN {X 0,Y 602.375,Z 853.653,A -85,B 0,C 180,E1 -7318.667,E2 -7318.667} C_VEL
LIN {X 0,Y 604.021,Z 832.771,A -85,B 0,C 180,E1 -7320.045,E2 -7320.045} C_VEL
LIN {X 0,Y 605.574,Z 811.745,A -85,B 0,C 180,E1 -7321.229,E2 -7321.229} C_VEL
LIN {X 0,Y 606.946,Z 791.26,A -85,B 0,C 180,E1 -7322.227,E2 -7322.227} C_VEL
LIN {X 0,Y 608.392,Z 766.811,A -85,B 0,C 180,E1 -7323.223,E2 -7323.223} C_VEL
LIN {X 0,Y 609.519,Z 745.309,A -85,B 0,C 180,E1 -7323.943,E2 -7323.943} C_VEL
LIN {X 0,Y 610.621,Z 720.009,A -85,B 0,C 180,E1 -7324.608,E2 -7324.608} C_VEL
LIN {X 0,Y 611.316,Z 699.017,A -85,B 0,C 180,E1 -7325.024,E2 -7325.024} C_VEL
LIN {X 0,Y 611.841,Z 665.599,A -85,B 0,C 180,E1 -7325.475,E2 -7325.475} C_VEL
LIN {X 0,Y 613.483,Z 505.056,A -85,B 0,C 180,E1 -7327.437,E2 -7327.437} C_VEL
LIN {X 0,Y 615.769,Z 370.353,A -85,B 0,C 180,E1 -7329.245,E2 -7329.245} C_VEL
LIN {X 0,Y 616.608,Z 325.242,A -85,B 0,C 180,E1 -7329.904,E2 -7329.904} C_VEL
LIN {X 0,Y 616.057,Z 320.097,A -85,B 0,C 180,E1 -7330.056,E2 -7330.056} C_VEL
LIN {X 0,Y 619.827,Z 294.353,A -85,B 0,C 180,E1 -7331.716,E2 -7331.716} C_VEL
LIN {X 0,Y 624.651,Z 271.49,A -85,B 0,C 180,E1 -7333.357,E2 -7333.357} C_VEL
LIN {X 0,Y 622.644,Z 264.81,A -85,B 0,C 180,E1 -7334.569,E2 -7334.569} C_VEL
LIN {X 0,Y 621.136,Z 260.554,A -85,B 0,C 180,E1 -7335.681,E2 -7335.681} C_VEL
LIN {X 0,Y 620.517,Z 258.704,A -85,B 0,C 180,E1 -7336.345,E2 -7336.345} C_VEL
LIN {X 0,Y 619.931,Z 256.317,A -85,B 0,C 180,E1 -7337.759,E2 -7337.759} C_VEL
LIN {X 0,Y 619.921,Z 256.156,A -85,B 0,C 180,E1 -7338.477,E2 -7338.477} C_VEL
LIN {X 0,Y 620.016,Z 258.169,A -85,B 0,C 180,E1 -7339.855,E2 -7339.855} C_VEL
LIN {X 0,Y 620.455,Z 259.852,A -85,B 0,C 180,E1 -7340.528,E2 -7340.528} C_VEL
LIN {X 0,Y 621.477,Z 263.67,A -85,B 0,C 180,E1 -7341.608,E2 -7341.608} C_VEL
LIN {X 0,Y 622.576,Z 268.976,A -85,B 0,C 180,E1 -7342.655,E2 -7342.655} C_VEL
LIN {X 0,Y 617.218,Z 291.995,A -85,B 0,C 180,E1 -7344.609,E2 -7344.609} C_VEL
LIN {X 0,Y 612.142,Z 323.112,A -85,B 0,C 180,E1 -7347.048,E2 -7347.048} C_VEL
LIN {X 0,Y 607.803,Z 361.756,A -85,B 0,C 180,E1 -7349.884,E2 -7349.884} C_VEL
LIN {X 0,Y 604.093,Z 407.305,A -85,B 0,C 180,E1 -7353.03,E2 -7353.03} C_VEL
LIN {X 0,Y 602.826,Z 429.307,A -85,B 0,C 180,E1 -7354.479,E2 -7354.479} C_VEL
LIN {X 0,Y 606.508,Z 463.394,A -85,B 0,C 180,E1 -7355.589,E2 -7355.589} C_VEL
LIN {X 0,Y 608.81,Z 491.541,A -85,B 0,C 180,E1 -7356.385,E2 -7356.385} C_VEL
LIN {X 0,Y 603.933,Z 594.04,A -85,B 0,C 180,E1 -7358.251,E2 -7358.251} C_VEL
LIN {X 0,Y 600.841,Z 686.375,A -85,B 0,C 180,E1 -7359.856,E2 -7359.856} C_VEL
LIN {X 0,Y 600.021,Z 708.486,A -85,B 0,C 180,E1 -7360.43,E2 -7360.43} C_VEL
LIN {X 0,Y 599.252,Z 728.145,A -85,B 0,C 180,E1 -7361.113,E2 -7361.113} C_VEL
LIN {X 0,Y 598.432,Z 746.855,A -85,B 0,C 180,E1 -7361.937,E2 -7361.937} C_VEL
LIN {X 0,Y 597.641,Z 764.094,A -85,B 0,C 180,E1 -7362.875,E2 -7362.875} C_VEL
LIN {X 0,Y 596.819,Z 781.182,A -85,B 0,C 180,E1 -7364.002,E2 -7364.002} C_VEL
LIN {X 0,Y 596.06,Z 795.961,A -85,B 0,C 180,E1 -7365.178,E2 -7365.178} C_VEL
LIN {X 0,Y 595.379,Z 808.862,A -85,B 0,C 180,E1 -7366.401,E2 -7366.401} C_VEL
LIN {X 0,Y 594.741,Z 820.979,A -85,B 0,C 180,E1 -7367.77,E2 -7367.77} C_VEL
LIN {X 0,Y 594.146,Z 832.402,A -85,B 0,C 180,E1 -7369.332,E2 -7369.332} C_VEL
LIN {X 0,Y 593.677,Z 841.64,A -85,B 0,C 180,E1 -7370.891,E2 -7370.891} C_VEL
LIN {X 0,Y 593.308,Z 849.424,A -85,B 0,C 180,E1 -7372.544,E2 -7372.544} C_VEL
LIN {X 0,Y 593.041,Z 855.653,A -85,B 0,C 180,E1 -7374.291,E2 -7374.291} C_VEL
LIN {X 0,Y 592.845,Z 860.031,A -85,B 0,C 180,E1 -7376.035,E2 -7376.035} C_VEL
LIN {X 0,Y 592.713,Z 862.766,A -85,B 0,C 180,E1 -7377.873,E2 -7377.873} C_VEL
LIN {X 0,Y 592.641,Z 863.646,A -85,B 0,C 180,E1 -7379.71,E2 -7379.71} C_VEL
LIN {X 0,Y 592.601,Z 862.707,A -85,B 0,C 180,E1 -7381.547,E2 -7381.547} C_VEL
LIN {X 0,Y 592.619,Z 859.957,A -85,B 0,C 180,E1 -7383.386,E2 -7383.386} C_VEL
LIN {X 0,Y 592.701,Z 855.339,A -85,B 0,C 180,E1 -7385.227,E2 -7385.227} C_VEL
LIN {X 0,Y 592.855,Z 849.127,A -85,B 0,C 180,E1 -7386.975,E2 -7386.975} C_VEL
LIN {X 0,Y 593.118,Z 840.959,A -85,B 0,C 180,E1 -7388.727,E2 -7388.727} C_VEL
LIN {X 0,Y 593.505,Z 831.215,A -85,B 0,C 180,E1 -7390.385,E2 -7390.385} C_VEL
LIN {X 0,Y 594.007,Z 819.939,A -85,B 0,C 180,E1 -7391.949,E2 -7391.949} C_VEL
LIN {X 0,Y 594.621,Z 807.123,A -85,B 0,C 180,E1 -7393.418,E2 -7393.418} C_VEL
LIN {X 0,Y 595.336,Z 792.725,A -85,B 0,C 180,E1 -7394.791,E2 -7394.791} C_VEL
LIN {X 0,Y 596.127,Z 777.057,A -85,B 0,C 180,E1 -7396.033,E2 -7396.033} C_VEL
LIN {X 0,Y 596.94,Z 760.104,A -85,B 0,C 180,E1 -7397.146,E2 -7397.146} C_VEL
LIN {X 0,Y 597.789,Z 741.744,A -85,B 0,C 180,E1 -7398.126,E2 -7398.126} C_VEL
LIN {X 0,Y 598.573,Z 723.368,A -85,B 0,C 180,E1 -7398.909,E2 -7398.909} C_VEL
LIN {X 0,Y 599.278,Z 703.626,A -85,B 0,C 180,E1 -7399.557,E2 -7399.557} C_VEL
LIN {X 0,Y 599.868,Z 683.691,A -85,B 0,C 180,E1 -7400.025,E2 -7400.025} C_VEL
LIN {X 0,Y 600.507,Z 648.006,A -85,B 0,C 180,E1 -7400.555,E2 -7400.555} C_VEL
LIN {X 0,Y 603.646,Z 487.791,A -85,B 0,C 180,E1 -7402.848,E2 -7402.848} C_VEL
LIN {X 0,Y 600.129,Z 457.216,A -85,B 0,C 180,E1 -7403.492,E2 -7403.492} C_VEL
LIN {X 0,Y 602.242,Z 407.046,A -85,B 0,C 180,E1 -7406.633,E2 -7406.633} C_VEL
LIN {X 0,Y 604.811,Z 353.862,A -85,B 0,C 180,E1 -7410.001,E2 -7410.001} C_VEL
LIN {X 0,Y 607.533,Z 300.915,A -85,B 0,C 180,E1 -7413.409,E2 -7413.409} C_VEL
LIN {X 0,Y 608.182,Z 289.748,A -85,B 0,C 180,E1 -7414.133,E2 -7414.133} C_VEL
LIN {X 0,Y 607.662,Z 283.643,A -85,B 0,C 180,E1 -7414.582,E2 -7414.582} C_VEL
LIN {X 0,Y 603.085,Z 268.41,A -85,B 0,C 180,E1 -7415.919,E2 -7415.919} C_VEL
LIN {X 0,Y 602.76,Z 263.158,A -85,B 0,C 180,E1 -7416.308,E2 -7416.308} C_VEL
LIN {X 0,Y 603,Z 258.062,A -85,B 0,C 180,E1 -7416.652,E2 -7416.652} C_VEL
LIN {X 0,Y 593.193,Z 232.341,A -85,B 0,C 180,E1 -7419.16,E2 -7419.16} C_VEL
LIN {X 0,Y 585.291,Z 212.68,A -85,B 0,C 180,E1 -7421.199,E2 -7421.199} C_VEL
LIN {X 0,Y 585.248,Z 212.328,A -85,B 0,C 180,E1 -7421.26,E2 -7421.26} C_VEL
LIN {X 0,Y 585.242,Z 212.33,A -85,B 0,C 180,E1 -7424.466,E2 -7424.466} C_VEL
LIN {X 0,Y 585.279,Z 212.511,A -85,B 0,C 180,E1 -7427.419,E2 -7427.419} C_VEL
LIN {X 0,Y 586.486,Z 215.688,A -85,B 0,C 180,E1 -7427.725,E2 -7427.725} C_VEL
LIN {X 0,Y 593.915,Z 231.577,A -85,B 0,C 180,E1 -7429.402,E2 -7429.402} C_VEL
LIN {X 0,Y 600.68,Z 248.052,A -85,B 0,C 180,E1 -7431.13,E2 -7431.13} C_VEL
LIN {X 0,Y 606.998,Z 264.685,A -85,B 0,C 180,E1 -7432.872,E2 -7432.872} C_VEL
LIN {X 0,Y 605.845,Z 307.892,A -85,B 0,C 180,E1 -7435.979,E2 -7435.979} C_VEL
LIN {X 0,Y 605.978,Z 335.125,A -85,B 0,C 180,E1 -7437.766,E2 -7437.766} C_VEL
LIN {X 0,Y 605.422,Z 338.502,A -85,B 0,C 180,E1 -7437.876,E2 -7437.876} C_VEL
LIN {X 0,Y 603.338,Z 437.852,A -85,B 0,C 180,E1 -7439.212,E2 -7439.212} C_VEL
LIN {X 0,Y 600.331,Z 537.417,A -85,B 0,C 180,E1 -7440.735,E2 -7440.735} C_VEL
LIN {X 0,Y 597.515,Z 624.806,A -85,B 0,C 180,E1 -7442.216,E2 -7442.216} C_VEL
LIN {X 0,Y 596.746,Z 647.196,A -85,B 0,C 180,E1 -7442.768,E2 -7442.768} C_VEL
LIN {X 0,Y 595.726,Z 669.58,A -85,B 0,C 180,E1 -7443.51,E2 -7443.51} C_VEL
LIN {X 0,Y 594.586,Z 690.638,A -85,B 0,C 180,E1 -7444.394,E2 -7444.394} C_VEL
LIN {X 0,Y 593.358,Z 710.362,A -85,B 0,C 180,E1 -7445.403,E2 -7445.403} C_VEL
LIN {X 0,Y 592.002,Z 729.982,A -85,B 0,C 180,E1 -7446.614,E2 -7446.614} C_VEL
LIN {X 0,Y 590.67,Z 747.957,A -85,B 0,C 180,E1 -7447.926,E2 -7447.926} C_VEL
LIN {X 0,Y 589.337,Z 765.647,A -85,B 0,C 180,E1 -7449.439,E2 -7449.439} C_VEL
LIN {X 0,Y 588.14,Z 781.742,A -85,B 0,C 180,E1 -7451.051,E2 -7451.051} C_VEL
LIN {X 0,Y 587.085,Z 796.378,A -85,B 0,C 180,E1 -7452.762,E2 -7452.762} C_VEL
LIN {X 0,Y 586.208,Z 809.56,A -85,B 0,C 180,E1 -7454.568,E2 -7454.568} C_VEL
LIN {X 0,Y 585.514,Z 820.562,A -85,B 0,C 180,E1 -7456.369,E2 -7456.369} C_VEL
LIN {X 0,Y 584.953,Z 830.748,A -85,B 0,C 180,E1 -7458.369,E2 -7458.369} C_VEL
LIN {X 0,Y 584.605,Z 838.635,A -85,B 0,C 180,E1 -7460.251,E2 -7460.251} C_VEL
LIN {X 0,Y 584.357,Z 845.109,A -85,B 0,C 180,E1 -7462.231,E2 -7462.231} C_VEL
LIN {X 0,Y 584.223,Z 850.242,A -85,B 0,C 180,E1 -7464.303,E2 -7464.303} C_VEL
LIN {X 0,Y 584.169,Z 853.792,A -85,B 0,C 180,E1 -7466.369,E2 -7466.369} C_VEL
LIN {X 0,Y 584.134,Z 855.693,A -85,B 0,C 180,E1 -7468.431,E2 -7468.431} C_VEL
LIN {X 0,Y 584.121,Z 856.094,A -85,B 0,C 180,E1 -7470.588,E2 -7470.588} C_VEL
LIN {X 0,Y 584.145,Z 854.987,A -85,B 0,C 180,E1 -7472.649,E2 -7472.649} C_VEL
LIN {X 0,Y 584.195,Z 852.266,A -85,B 0,C 180,E1 -7474.712,E2 -7474.712} C_VEL
LIN {X 0,Y 584.275,Z 847.985,A -85,B 0,C 180,E1 -7476.781,E2 -7476.781} C_VEL
LIN {X 0,Y 584.455,Z 842.401,A -85,B 0,C 180,E1 -7478.758,E2 -7478.758} C_VEL
LIN {X 0,Y 584.77,Z 835.046,A -85,B 0,C 180,E1 -7480.741,E2 -7480.741} C_VEL
LIN {X 0,Y 585.214,Z 825.867,A -85,B 0,C 180,E1 -7482.733,E2 -7482.733} C_VEL
LIN {X 0,Y 585.834,Z 815.242,A -85,B 0,C 180,E1 -7484.632,E2 -7484.632} C_VEL
LIN {X 0,Y 586.629,Z 803.187,A -85,B 0,C 180,E1 -7486.436,E2 -7486.436} C_VEL
LIN {X 0,Y 587.629,Z 788.821,A -85,B 0,C 180,E1 -7488.245,E2 -7488.245} C_VEL
LIN {X 0,Y 588.721,Z 773.876,A -85,B 0,C 180,E1 -7489.857,E2 -7489.857} C_VEL
LIN {X 0,Y 589.989,Z 756.998,A -85,B 0,C 180,E1 -7491.421,E2 -7491.421} C_VEL
LIN {X 0,Y 591.287,Z 739.838,A -85,B 0,C 180,E1 -7492.783,E2 -7492.783} C_VEL
LIN {X 0,Y 592.627,Z 721.224,A -85,B 0,C 180,E1 -7494.046,E2 -7494.046} C_VEL
LIN {X 0,Y 593.978,Z 700.668,A -85,B 0,C 180,E1 -7495.207,E2 -7495.207} C_VEL
LIN {X 0,Y 595.117,Z 681.189,A -85,B 0,C 180,E1 -7496.117,E2 -7496.117} C_VEL
LIN {X 0,Y 596.2,Z 659.94,A -85,B 0,C 180,E1 -7496.925,E2 -7496.925} C_VEL
LIN {X 0,Y 597.08,Z 638.557,A -85,B 0,C 180,E1 -7497.559,E2 -7497.559} C_VEL
LIN {X 0,Y 597.784,Z 616.015,A -85,B 0,C 180,E1 -7498.046,E2 -7498.046} C_VEL
LIN {X 0,Y 601.653,Z 496.299,A -85,B 0,C 180,E1 -7500.005,E2 -7500.005} C_VEL
LIN {X 0,Y 604.151,Z 405.264,A -85,B 0,C 180,E1 -7501.336,E2 -7501.336} C_VEL
LIN {X 0,Y 605.491,Z 337.381,A -85,B 0,C 180,E1 -7502.235,E2 -7502.235} C_VEL
LIN {X 0,Y 605.977,Z 334.126,A -85,B 0,C 180,E1 -7502.39,E2 -7502.39} C_VEL
LIN {X 0,Y 605.917,Z 305.223,A -85,B 0,C 180,E1 -7504.301,E2 -7504.301} C_VEL
LIN {X 0,Y 606.972,Z 264.587,A -85,B 0,C 180,E1 -7507.236,E2 -7507.236} C_VEL
LIN {X 0,Y 598.693,Z 242.855,A -85,B 0,C 180,E1 -7509.518,E2 -7509.518} C_VEL
LIN {X 0,Y 590.816,Z 224.56,A -85,B 0,C 180,E1 -7511.433,E2 -7511.433} C_VEL
LIN {X 0,Y 586.342,Z 215.469,A -85,B 0,C 180,E1 -7512.405,E2 -7512.405} C_VEL
LIN {X 0,Y 585.243,Z 212.329,A -85,B 0,C 180,E1 -7512.721,E2 -7512.721} C_VEL
LIN {X 0,Y 585.253,Z 212.321,A -85,B 0,C 180,E1 -7515.994,E2 -7515.994} C_VEL
LIN {X 0,Y 585.234,Z 212.324,A -85,B 0,C 180,E1 -7519.19,E2 -7519.19} C_VEL
LIN {X 0,Y 585.255,Z 212.32,A -85,B 0,C 180,E1 -7522.441,E2 -7522.441} C_VEL
LIN {X 0,Y 585.254,Z 212.324,A -85,B 0,C 180,E1 -7525.8,E2 -7525.8} C_VEL
LIN {X 0,Y 585.241,Z 212.328,A -85,B 0,C 180,E1 -7529.056,E2 -7529.056} C_VEL
LIN {X 0,Y 585.247,Z 212.317,A -85,B 0,C 180,E1 -7532.308,E2 -7532.308} C_VEL
LIN {X 0,Y 585.251,Z 212.313,A -85,B 0,C 180,E1 -7535.591,E2 -7535.591} C_VEL
LIN {X 0,Y 585.253,Z 212.323,A -85,B 0,C 180,E1 -7538.975,E2 -7538.975} C_VEL
LIN {X 0,Y 585.241,Z 212.306,A -85,B 0,C 180,E1 -7542.192,E2 -7542.192} C_VEL
LIN {X 0,Y 585.249,Z 212.328,A -85,B 0,C 180,E1 -7545.454,E2 -7545.454} C_VEL
LIN {X 0,Y 585.249,Z 212.311,A -85,B 0,C 180,E1 -7548.769,E2 -7548.769} C_VEL
LIN {X 0,Y 585.244,Z 212.321,A -85,B 0,C 180,E1 -7552.045,E2 -7552.045} C_VEL
LIN {X 0,Y 585.249,Z 212.31,A -85,B 0,C 180,E1 -7555.296,E2 -7555.296} C_VEL
LIN {X 0,Y 585.235,Z 212.322,A -85,B 0,C 180,E1 -7558.531,E2 -7558.531} C_VEL
LIN {X 0,Y 585.253,Z 212.307,A -85,B 0,C 180,E1 -7561.762,E2 -7561.762} C_VEL
LIN {X 0,Y 585.255,Z 212.323,A -85,B 0,C 180,E1 -7565.102,E2 -7565.102} C_VEL
LIN {X 0,Y 585.226,Z 212.316,A -85,B 0,C 180,E1 -7568.35,E2 -7568.35} C_VEL
LIN {X 0,Y 585.257,Z 212.329,A -85,B 0,C 180,E1 -7571.531,E2 -7571.531} C_VEL
LIN {X 0,Y 585.23,Z 212.325,A -85,B 0,C 180,E1 -7574.752,E2 -7574.752} C_VEL
LIN {X 0,Y 585.238,Z 212.326,A -85,B 0,C 180,E1 -7578.117,E2 -7578.117} C_VEL
LIN {X 0,Y 585.261,Z 212.324,A -85,B 0,C 180,E1 -7581.34,E2 -7581.34} C_VEL
LIN {X 0,Y 585.219,Z 212.33,A -85,B 0,C 180,E1 -7584.531,E2 -7584.531} C_VEL
LIN {X 0,Y 585.262,Z 212.327,A -85,B 0,C 180,E1 -7587.751,E2 -7587.751} C_VEL
LIN {X 0,Y 585.224,Z 212.33,A -85,B 0,C 180,E1 -7590.949,E2 -7590.949} C_VEL
LIN {X 0,Y 585.222,Z 212.33,A -85,B 0,C 180,E1 -7594.321,E2 -7594.321} C_VEL
LIN {X 0,Y 585.257,Z 212.326,A -85,B 0,C 180,E1 -7597.461,E2 -7597.461} C_VEL
LIN {X 0,Y 585.261,Z 212.338,A -85,B 0,C 180,E1 -7599.906,E2 -7599.906} C_VEL
LIN {X 0,Y 586.381,Z 215.581,A -85,B 0,C 180,E1 -7600.261,E2 -7600.261} C_VEL
LIN {X 0,Y 587.608,Z 217.746,A -85,B 0,C 180,E1 -7600.543,E2 -7600.543} C_VEL
LIN {X 0,Y 598.082,Z 238.251,A -85,B 0,C 180,E1 -7603.009,E2 -7603.009} C_VEL
LIN {X 0,Y 610.673,Z 263.873,A -85,B 0,C 180,E1 -7605.821,E2 -7605.821} C_VEL
LIN {X 0,Y 614.414,Z 272.176,A -85,B 0,C 180,E1 -7606.658,E2 -7606.658} C_VEL
LIN {X 0,Y 611.616,Z 308.131,A -85,B 0,C 180,E1 -7608.624,E2 -7608.624} C_VEL
LIN {X 0,Y 614.335,Z 329.922,A -85,B 0,C 180,E1 -7609.152,E2 -7609.152} C_VEL
LIN {X 0,Y 609.104,Z 573.453,A -85,B 0,C 180,E1 -7612.47,E2 -7612.47} C_VEL
LIN {X 0,Y 606.877,Z 692.706,A -85,B 0,C 180,E1 -7614.055,E2 -7614.055} C_VEL
LIN {X 0,Y 605.881,Z 717.138,A -85,B 0,C 180,E1 -7614.54,E2 -7614.54} C_VEL
LIN {X 0,Y 604.759,Z 738.145,A -85,B 0,C 180,E1 -7615.09,E2 -7615.09} C_VEL
LIN {X 0,Y 603.156,Z 763.07,A -85,B 0,C 180,E1 -7615.922,E2 -7615.922} C_VEL
LIN {X 0,Y 601.633,Z 783.135,A -85,B 0,C 180,E1 -7616.74,E2 -7616.74} C_VEL
LIN {X 0,Y 599.724,Z 806.743,A -85,B 0,C 180,E1 -7617.883,E2 -7617.883} C_VEL
LIN {X 0,Y 597.919,Z 827.166,A -85,B 0,C 180,E1 -7619.054,E2 -7619.054} C_VEL
LIN {X 0,Y 595.794,Z 849.632,A -85,B 0,C 180,E1 -7620.546,E2 -7620.546} C_VEL
LIN {X 0,Y 593.972,Z 868.39,A -85,B 0,C 180,E1 -7621.987,E2 -7621.987} C_VEL
LIN {X 0,Y 592.002,Z 888.828,A -85,B 0,C 180,E1 -7623.789,E2 -7623.789} C_VEL
LIN {X 0,Y 590.374,Z 905.637,A -85,B 0,C 180,E1 -7625.484,E2 -7625.484} C_VEL
LIN {X 0,Y 588.74,Z 923.368,A -85,B 0,C 180,E1 -7627.534,E2 -7627.534} C_VEL
LIN {X 0,Y 587.493,Z 937.528,A -85,B 0,C 180,E1 -7629.404,E2 -7629.404} C_VEL
LIN {X 0,Y 586.327,Z 952.004,A -85,B 0,C 180,E1 -7631.61,E2 -7631.61} C_VEL
LIN {X 0,Y 585.634,Z 961.798,A -85,B 0,C 180,E1 -7633.331,E2 -7633.331} C_VEL
LIN {X 0,Y 584.963,Z 971.848,A -85,B 0,C 180,E1 -7635.447,E2 -7635.447} C_VEL
LIN {X 0,Y 584.459,Z 980.895,A -85,B 0,C 180,E1 -7637.752,E2 -7637.752} C_VEL
LIN {X 0,Y 584.169,Z 987.725,A -85,B 0,C 180,E1 -7639.846,E2 -7639.846} C_VEL
LIN {X 0,Y 583.971,Z 994.069,A -85,B 0,C 180,E1 -7642.325,E2 -7642.325} C_VEL
LIN {X 0,Y 583.92,Z 997.973,A -85,B 0,C 180,E1 -7644.399,E2 -7644.399} C_VEL
LIN {X 0,Y 583.898,Z 1001.016,A -85,B 0,C 180,E1 -7646.761,E2 -7646.761} C_VEL
LIN {X 0,Y 583.897,Z 1002.28,A -85,B 0,C 180,E1 -7649.019,E2 -7649.019} C_VEL
LIN {X 0,Y 583.896,Z 1002.28,A -85,B 0,C 180,E1 -7650.981,E2 -7650.981} C_VEL
LIN {X 0,Y 583.902,Z 1000.914,A -85,B 0,C 180,E1 -7653.338,E2 -7653.338} C_VEL
LIN {X 0,Y 583.92,Z 997.971,A -85,B 0,C 180,E1 -7655.601,E2 -7655.601} C_VEL
LIN {X 0,Y 583.972,Z 994.069,A -85,B 0,C 180,E1 -7657.675,E2 -7657.675} C_VEL
LIN {X 0,Y 584.174,Z 987.581,A -85,B 0,C 180,E1 -7660.201,E2 -7660.201} C_VEL
LIN {X 0,Y 584.459,Z 980.893,A -85,B 0,C 180,E1 -7662.248,E2 -7662.248} C_VEL
LIN {X 0,Y 584.963,Z 971.848,A -85,B 0,C 180,E1 -7664.553,E2 -7664.553} C_VEL
LIN {X 0,Y 585.635,Z 961.803,A -85,B 0,C 180,E1 -7666.669,E2 -7666.669} C_VEL
LIN {X 0,Y 586.237,Z 953.139,A -85,B 0,C 180,E1 -7668.19,E2 -7668.19} C_VEL
LIN {X 0,Y 587.284,Z 939.88,A -85,B 0,C 180,E1 -7670.22,E2 -7670.22} C_VEL
LIN {X 0,Y 588.481,Z 924.956,A -85,B 0,C 180,E1 -7672.178,E2 -7672.178} C_VEL
LIN {X 0,Y 589.851,Z 909.137,A -85,B 0,C 180,E1 -7674.006,E2 -7674.006} C_VEL
LIN {X 0,Y 591.407,Z 891.183,A -85,B 0,C 180,E1 -7675.808,E2 -7675.808} C_VEL
LIN {X 0,Y 593.018,Z 873.034,A -85,B 0,C 180,E1 -7677.407,E2 -7677.407} C_VEL
LIN {X 0,Y 594.747,Z 852.69,A -85,B 0,C 180,E1 -7678.959,E2 -7678.959} C_VEL
LIN {X 0,Y 596.345,Z 833.289,A -85,B 0,C 180,E1 -7680.255,E2 -7680.255} C_VEL
LIN {X 0,Y 598.015,Z 811.764,A -85,B 0,C 180,E1 -7681.49,E2 -7681.49} C_VEL
LIN {X 0,Y 599.428,Z 791.633,A -85,B 0,C 180,E1 -7682.488,E2 -7682.488} C_VEL
LIN {X 0,Y 601.005,Z 766.513,A -85,B 0,C 180,E1 -7683.528,E2 -7683.528} C_VEL
LIN {X 0,Y 602.239,Z 744.264,A -85,B 0,C 180,E1 -7684.282,E2 -7684.282} C_VEL
LIN {X 0,Y 603.361,Z 719.506,A -85,B 0,C 180,E1 -7684.936,E2 -7684.936} C_VEL
LIN {X 0,Y 604.09,Z 698.59,A -85,B 0,C 180,E1 -7685.355,E2 -7685.355} C_VEL
LIN {X 0,Y 604.653,Z 664.91,A -85,B 0,C 180,E1 -7685.815,E2 -7685.815} C_VEL
LIN {X 0,Y 606.419,Z 513.799,A -85,B 0,C 180,E1 -7687.697,E2 -7687.697} C_VEL
LIN {X 0,Y 608.891,Z 383.836,A -85,B 0,C 180,E1 -7689.481,E2 -7689.481} C_VEL
LIN {X 0,Y 610.213,Z 326.648,A -85,B 0,C 180,E1 -7690.34,E2 -7690.34} C_VEL
LIN {X 0,Y 609.782,Z 322.554,A -85,B 0,C 180,E1 -7690.461,E2 -7690.461} C_VEL
LIN {X 0,Y 613.985,Z 297.393,A -85,B 0,C 180,E1 -7692.141,E2 -7692.141} C_VEL
LIN {X 0,Y 619.057,Z 276.157,A -85,B 0,C 180,E1 -7693.701,E2 -7693.701} C_VEL
LIN {X 0,Y 617.446,Z 270.406,A -85,B 0,C 180,E1 -7694.822,E2 -7694.822} C_VEL
LIN {X 0,Y 616.157,Z 266.128,A -85,B 0,C 180,E1 -7696.008,E2 -7696.008} C_VEL
LIN {X 0,Y 615.288,Z 263.382,A -85,B 0,C 180,E1 -7697.405,E2 -7697.405} C_VEL
LIN {X 0,Y 615.355,Z 262.551,A -85,B 0,C 180,E1 -7698.231,E2 -7698.231} C_VEL
LIN {X 0,Y 615.239,Z 264.441,A -85,B 0,C 180,E1 -7699.697,E2 -7699.697} C_VEL
LIN {X 0,Y 615.563,Z 265.9,A -85,B 0,C 180,E1 -7700.349,E2 -7700.349} C_VEL
LIN {X 0,Y 616.38,Z 269.551,A -85,B 0,C 180,E1 -7701.435,E2 -7701.435} C_VEL
LIN {X 0,Y 617.125,Z 273.642,A -85,B 0,C 180,E1 -7702.292,E2 -7702.292} C_VEL
LIN {X 0,Y 611.54,Z 295.137,A -85,B 0,C 180,E1 -7704.173,E2 -7704.173} C_VEL
LIN {X 0,Y 606.196,Z 324.086,A -85,B 0,C 180,E1 -7706.513,E2 -7706.513} C_VEL
LIN {X 0,Y 601.464,Z 361.147,A -85,B 0,C 180,E1 -7709.312,E2 -7709.312} C_VEL
LIN {X 0,Y 597.304,Z 406.578,A -85,B 0,C 180,E1 -7712.527,E2 -7712.527} C_VEL
LIN {X 0,Y 596.036,Z 426.295,A -85,B 0,C 180,E1 -7713.851,E2 -7713.851} C_VEL
LIN {X 0,Y 599.748,Z 461.707,A -85,B 0,C 180,E1 -7715.061,E2 -7715.061} C_VEL
LIN {X 0,Y 602.193,Z 492.466,A -85,B 0,C 180,E1 -7715.967,E2 -7715.967} C_VEL
LIN {X 0,Y 596.686,Z 600.228,A -85,B 0,C 180,E1 -7717.989,E2 -7717.989} C_VEL
LIN {X 0,Y 593.541,Z 686.878,A -85,B 0,C 180,E1 -7719.546,E2 -7719.546} C_VEL
LIN {X 0,Y 592.663,Z 709.153,A -85,B 0,C 180,E1 -7720.135,E2 -7720.135} C_VEL
LIN {X 0,Y 591.792,Z 729.638,A -85,B 0,C 180,E1 -7720.866,E2 -7720.866} C_VEL
LIN {X 0,Y 590.868,Z 749.261,A -85,B 0,C 180,E1 -7721.756,E2 -7721.756} C_VEL
LIN {X 0,Y 590.016,Z 766.959,A -85,B 0,C 180,E1 -7722.748,E2 -7722.748} C_VEL
LIN {X 0,Y 589.169,Z 783.254,A -85,B 0,C 180,E1 -7723.857,E2 -7723.857} C_VEL
LIN {X 0,Y 588.317,Z 798.784,A -85,B 0,C 180,E1 -7725.129,E2 -7725.129} C_VEL
LIN {X 0,Y 587.535,Z 812.852,A -85,B 0,C 180,E1 -7726.517,E2 -7726.517} C_VEL
LIN {X 0,Y 586.836,Z 825.27,A -85,B 0,C 180,E1 -7728.002,E2 -7728.002} C_VEL
LIN {X 0,Y 586.228,Z 836.085,A -85,B 0,C 180,E1 -7729.584,E2 -7729.584} C_VEL
LIN {X 0,Y 585.724,Z 845.362,A -85,B 0,C 180,E1 -7731.27,E2 -7731.27} C_VEL
LIN {X 0,Y 585.36,Z 852.612,A -85,B 0,C 180,E1 -7732.953,E2 -7732.953} C_VEL
LIN {X 0,Y 585.097,Z 858.237,A -85,B 0,C 180,E1 -7734.705,E2 -7734.705} C_VEL
LIN {X 0,Y 584.899,Z 862.098,A -85,B 0,C 180,E1 -7736.472,E2 -7736.472} C_VEL
LIN {X 0,Y 584.764,Z 864.292,A -85,B 0,C 180,E1 -7738.334,E2 -7738.334} C_VEL
LIN {X 0,Y 584.702,Z 864.684,A -85,B 0,C 180,E1 -7740.098,E2 -7740.098} C_VEL
LIN {X 0,Y 584.671,Z 863.3,A -85,B 0,C 180,E1 -7741.96,E2 -7741.96} C_VEL
LIN {X 0,Y 584.698,Z 860.087,A -85,B 0,C 180,E1 -7743.824,E2 -7743.824} C_VEL
LIN {X 0,Y 584.801,Z 855.3,A -85,B 0,C 180,E1 -7745.593,E2 -7745.593} C_VEL
LIN {X 0,Y 584.974,Z 848.69,A -85,B 0,C 180,E1 -7747.365,E2 -7747.365} C_VEL
LIN {X 0,Y 585.275,Z 840.066,A -85,B 0,C 180,E1 -7749.142,E2 -7749.142} C_VEL
LIN {X 0,Y 585.712,Z 829.836,A -85,B 0,C 180,E1 -7750.824,E2 -7750.824} C_VEL
LIN {X 0,Y 586.274,Z 818.03,A -85,B 0,C 180,E1 -7752.409,E2 -7752.409} C_VEL
LIN {X 0,Y 586.985,Z 804.127,A -85,B 0,C 180,E1 -7753.948,E2 -7753.948} C_VEL
LIN {X 0,Y 587.785,Z 789.01,A -85,B 0,C 180,E1 -7755.334,E2 -7755.334} C_VEL
LIN {X 0,Y 588.613,Z 773.301,A -85,B 0,C 180,E1 -7756.531,E2 -7756.531} C_VEL
LIN {X 0,Y 589.473,Z 755.981,A -85,B 0,C 180,E1 -7757.625,E2 -7757.625} C_VEL
LIN {X 0,Y 590.364,Z 737.587,A -85,B 0,C 180,E1 -7758.567,E2 -7758.567} C_VEL
LIN {X 0,Y 591.164,Z 718.702,A -85,B 0,C 180,E1 -7759.333,E2 -7759.333} C_VEL
LIN {X 0,Y 591.869,Z 698.765,A -85,B 0,C 180,E1 -7759.944,E2 -7759.944} C_VEL
LIN {X 0,Y 592.457,Z 678.561,A -85,B 0,C 180,E1 -7760.377,E2 -7760.377} C_VEL
LIN {X 0,Y 596.329,Z 488.725,A -85,B 0,C 180,E1 -7763.149,E2 -7763.149} C_VEL
LIN {X 0,Y 592.66,Z 456.622,A -85,B 0,C 180,E1 -7763.833,E2 -7763.833} C_VEL
LIN {X 0,Y 594.885,Z 406.758,A -85,B 0,C 180,E1 -7766.989,E2 -7766.989} C_VEL
LIN {X 0,Y 597.647,Z 352.544,A -85,B 0,C 180,E1 -7770.46,E2 -7770.46} C_VEL
LIN {X 0,Y 600.505,Z 300.475,A -85,B 0,C 180,E1 -7773.847,E2 -7773.847} C_VEL
LIN {X 0,Y 602.76,Z 263.158,A -85,B 0,C 180,E1 -7776.308,E2 -7776.308} C_VEL
LIN {X 0,Y 602.249,Z 260.454,A -85,B 0,C 180,E1 -7776.531,E2 -7776.531} C_VEL
LIN {X 0,Y 599.563,Z 257.226,A -85,B 0,C 180,E1 -7776.933,E2 -7776.933} C_VEL
LIN {X 0,Y 593.361,Z 252.549,A -85,B 0,C 180,E1 -7777.676,E2 -7777.676} C_VEL
LIN {X 0,Y 591.877,Z 250.242,A -85,B 0,C 180,E1 -7777.944,E2 -7777.944} C_VEL
LIN {X 0,Y 582.778,Z 227.034,A -85,B 0,C 180,E1 -7780.303,E2 -7780.303} C_VEL
LIN {X 0,Y 577.284,Z 213.321,A -85,B 0,C 180,E1 -7781.791,E2 -7781.791} C_VEL
LIN {X 0,Y 577.318,Z 213.312,A -85,B 0,C 180,E1 -7784.962,E2 -7784.962} C_VEL
LIN {X 0,Y 577.306,Z 213.326,A -85,B 0,C 180,E1 -7786.77,E2 -7786.77} C_VEL
LIN {X 0,Y 578.39,Z 216.458,A -85,B 0,C 180,E1 -7787.068,E2 -7787.068} C_VEL
LIN {X 0,Y 579.741,Z 219.06,A -85,B 0,C 180,E1 -7787.358,E2 -7787.358} C_VEL
LIN {X 0,Y 587.775,Z 236.28,A -85,B 0,C 180,E1 -7789.202,E2 -7789.202} C_VEL
LIN {X 0,Y 595.769,Z 256.018,A -85,B 0,C 180,E1 -7791.299,E2 -7791.299} C_VEL
LIN {X 0,Y 600.354,Z 268.408,A -85,B 0,C 180,E1 -7792.603,E2 -7792.603} C_VEL
LIN {X 0,Y 599.285,Z 311.246,A -85,B 0,C 180,E1 -7795.671,E2 -7795.671} C_VEL
LIN {X 0,Y 599.439,Z 336.798,A -85,B 0,C 180,E1 -7797.343,E2 -7797.343} C_VEL
LIN {X 0,Y 598.667,Z 341.014,A -85,B 0,C 180,E1 -7797.492,E2 -7797.492} C_VEL
LIN {X 0,Y 596.521,Z 438.755,A -85,B 0,C 180,E1 -7798.819,E2 -7798.819} C_VEL
LIN {X 0,Y 593.543,Z 532.789,A -85,B 0,C 180,E1 -7800.277,E2 -7800.277} C_VEL
LIN {X 0,Y 590.364,Z 624.995,A -85,B 0,C 180,E1 -7801.869,E2 -7801.869} C_VEL
LIN {X 0,Y 589.56,Z 647.957,A -85,B 0,C 180,E1 -7802.437,E2 -7802.437} C_VEL
LIN {X 0,Y 588.536,Z 669.721,A -85,B 0,C 180,E1 -7803.16,E2 -7803.16} C_VEL
LIN {X 0,Y 587.392,Z 690.277,A -85,B 0,C 180,E1 -7804.023,E2 -7804.023} C_VEL
LIN {X 0,Y 586.04,Z 710.662,A -85,B 0,C 180,E1 -7805.075,E2 -7805.075} C_VEL
LIN {X 0,Y 584.669,Z 729.58,A -85,B 0,C 180,E1 -7806.25,E2 -7806.25} C_VEL
LIN {X 0,Y 583.248,Z 747.753,A -85,B 0,C 180,E1 -7807.577,E2 -7807.577} C_VEL
LIN {X 0,Y 581.878,Z 765.048,A -85,B 0,C 180,E1 -7809.058,E2 -7809.058} C_VEL
LIN {X 0,Y 580.654,Z 780.427,A -85,B 0,C 180,E1 -7810.589,E2 -7810.589} C_VEL
LIN {X 0,Y 579.482,Z 795.245,A -85,B 0,C 180,E1 -7812.321,E2 -7812.321} C_VEL
LIN {X 0,Y 578.55,Z 807.897,A -85,B 0,C 180,E1 -7814.05,E2 -7814.05} C_VEL
LIN {X 0,Y 577.748,Z 819.913,A -85,B 0,C 180,E1 -7815.978,E2 -7815.978} C_VEL
LIN {X 0,Y 577.166,Z 829.985,A -85,B 0,C 180,E1 -7817.9,E2 -7817.9} C_VEL
LIN {X 0,Y 576.749,Z 838.161,A -85,B 0,C 180,E1 -7819.815,E2 -7819.815} C_VEL
LIN {X 0,Y 576.472,Z 845.031,A -85,B 0,C 180,E1 -7821.823,E2 -7821.823} C_VEL
LIN {X 0,Y 576.332,Z 850.343,A -85,B 0,C 180,E1 -7823.825,E2 -7823.825} C_VEL
LIN {X 0,Y 576.238,Z 854.154,A -85,B 0,C 180,E1 -7825.92,E2 -7825.92} C_VEL
LIN {X 0,Y 576.207,Z 856.482,A -85,B 0,C 180,E1 -7828.111,E2 -7828.111} C_VEL
LIN {X 0,Y 576.199,Z 857.182,A -85,B 0,C 180,E1 -7830.199,E2 -7830.199} C_VEL
LIN {X 0,Y 576.204,Z 856.281,A -85,B 0,C 180,E1 -7832.287,E2 -7832.287} C_VEL
